        (* Switch: '<S1>/Switch2' incorporates:
         *  Constant: '<S1>/Constant3' *)

        IF Enable THEN 
            (* Switch: '<S1>/Switch3' incorporates:
             *  Constant: '<S1>/Constant3'
             *  Gain: '<S1>/Gain'
             *  Gain: '<S1>/Gain3'
             *  Gain: '<S1>/muC'
             *  Product: '<S1>/Product'
             *  Product: '<S1>/Product1'
             *  Sum: '<S1>/Add'
             *  Sum: '<S1>/Subtract'
             *  Sum: '<S1>/Subtract1' *)

            IF Clock > 0.01 THEN 
                uPF := ((((pAsimbar - pp) * 100000.0) - (((pBsimbar - pr) * 100000.0) * 0.7101)) * HPF_Num1) * kQf;
            ELSE 
                uPF := 0.0;
            END_IF;

            (* End of Switch: '<S1>/Switch3' *)
        ELSE 
            uPF := 0.0;
        END_IF;

        (* End of Switch: '<S1>/Switch2' *)
        

        (* Saturate: '<S1>/Saturation5' *)

        IF uPF >= 3600.0 THEN 
            uPF := 3600.0;
        ELSIF uPF <= -3600.0 THEN 
            uPF := -3600.0;
        END_IF;

        (* End of Saturate: '<S1>/Saturation5' *)
END_CASE;

END_FUNCTION_BLOCK

// IndraMotionMlc1/Application/SCC_Acceleration_Feedback
FUNCTION_BLOCK SCC_Acceleration_Feedback
VAR_INPUT
	ssMethodType: SINT;
	AF_on: BOOL;
	Direct_on: BOOL;
	LPF_on: BOOL;
	HPF_on: BOOL;
	Acc_Input: LREAL;
	D_rev: LREAL;
	K_Direct: LREAL;
	LPF_Num1: LREAL;
	LPF_Num2: LREAL;
	LPF_Den1: LREAL;
	LPF_Den2: LREAL;
	HPF_Num1: LREAL;
	HPF_Num2: LREAL;
	HPF_Den1: LREAL;
	HPF_Den2: LREAL;
	b_reset: BOOL;
END_VAR
VAR_OUTPUT
	u_Direct: LREAL;
	u_LPF: LREAL;
	u_HPF: LREAL;
	u_AF: LREAL;
END_VAR
VAR
	rtb_DiscreteTransferFcn: LREAL;
	rtb_DiscreteTransferFcn1: LREAL;
	rtb_bDirect: LREAL;
	rtb_bLPF: LREAL;
	rtb_bHPF: DINT;
	DiscreteTransferFcn_tmp: LREAL;
	tmp: BOOL;
	temp1: BOOL;
	temp2: BOOL;
	VectorConcatenate: ARRAY[0..1] OF LREAL;
	VectorConcatenate1: ARRAY[0..1] OF LREAL;
	VectorConcatenate2: ARRAY[0..1] OF LREAL;
	VectorConcatenate3: ARRAY[0..1] OF LREAL;
	DiscreteTransferFcn_states: LREAL;
	DiscreteTransferFcn1_states: LREAL;
END_VAR



CASE ssMethodType OF
    0: 
        (* SystemInitialize for Atomic SubSystem: '<Root>/SCC_Acceleration_Feedback' *)
        (* InitializeConditions for DiscreteTransferFcn: '<S1>/Discrete Transfer Fcn' *)
        DiscreteTransferFcn_states := 0.0;
        (* InitializeConditions for DiscreteTransferFcn: '<S1>/Discrete Transfer Fcn1' *)
        DiscreteTransferFcn1_states := 0.0;
        (* End of SystemInitialize for SubSystem: '<Root>/SCC_Acceleration_Feedback' *)
    1: 
        (* Outputs for Atomic SubSystem: '<Root>/SCC_Acceleration_Feedback' *)
        (* SignalConversion: '<S1>/ConcatBufferAtVector ConcatenateIn1' *)
        VectorConcatenate[0] := HPF_Num1;
        (* SignalConversion: '<S1>/ConcatBufferAtVector ConcatenateIn2' *)
        VectorConcatenate[1] := HPF_Num2;
        (* SignalConversion: '<S1>/ConcatBufferAtVector Concatenate1In1' *)
        VectorConcatenate1[0] := HPF_Den1;
        (* SignalConversion: '<S1>/ConcatBufferAtVector Concatenate1In2' *)
        VectorConcatenate1[1] := HPF_Den2;
        (* SignalConversion: '<S1>/ConcatBufferAtVector Concatenate2In1' *)
        VectorConcatenate2[0] := LPF_Num1;
        (* SignalConversion: '<S1>/ConcatBufferAtVector Concatenate2In2' *)
        VectorConcatenate2[1] := LPF_Num2;
        (* SignalConversion: '<S1>/ConcatBufferAtVector Concatenate3In1' *)
        VectorConcatenate3[0] := LPF_Den1;
        (* SignalConversion: '<S1>/ConcatBufferAtVector Concatenate3In2' *)
        VectorConcatenate3[1] := LPF_Den2;
        (* Product: '<S1>/Divide' incorporates:
         *  Gain: '<S1>/Unit Gain2'
         *  Product: '<S1>/Product' *)
        u_Direct := ((K_Direct * Acc_Input) * 6.0E+7) / D_rev;
        (* MATLAB Function: '<S1>/MATLAB Function' *)
        (* MATLAB Function 'SCC_Acceleration_Feedback/MATLAB Function': '<S2>:1' *)
        (* '<S2>:1:3' bDirect = 0; *)
        rtb_bDirect := 0.0;
        (* '<S2>:1:4' bLPF = 0; *)
        rtb_bLPF := 0.0;
        (* '<S2>:1:5' bHPF = 0; *)
        rtb_bHPF := 0;
        (* '<S2>:1:7' if Direct_on == 1 &amp;&amp; LPF_on == 0 &amp;&amp; HPF_on == 0 *)
        tmp :=  NOT HPF_on;
        temp2 :=  NOT LPF_on;

        IF (Direct_on AND temp2) AND tmp THEN 
            (* '<S2>:1:8' bDirect = 1; *)
            rtb_bDirect := 1.0;
        ELSE 
            temp1 :=  NOT Direct_on;

            IF (temp1 AND LPF_on) AND tmp THEN 
                (* '<S2>:1:9' elseif Direct_on == 0 &amp;&amp; LPF_on == 1 &amp;&amp; HPF_on == 0 *)
                (* '<S2>:1:10' bLPF = 1; *)
                rtb_bLPF := 1.0;
            ELSIF (temp1 AND temp2) AND HPF_on THEN 
                (* '<S2>:1:11' elseif Direct_on == 0 &amp;&amp; LPF_on == 0 &amp;&amp; HPF_on == 1 *)
                (* '<S2>:1:12' bHPF = 1; *)
                rtb_bHPF := 1;
            END_IF;

        END_IF;

        (* End of MATLAB Function: '<S1>/MATLAB Function' *)
        

        (* DiscreteTransferFcn: '<S1>/Discrete Transfer Fcn' incorporates:
         *  DiscreteTransferFcn: '<S1>/Discrete Transfer Fcn1' *)

        IF b_reset THEN 
            DiscreteTransferFcn_states := 0.0;
            DiscreteTransferFcn1_states := 0.0;
        END_IF;

        DiscreteTransferFcn_tmp := Acc_Input - (VectorConcatenate3[1] * DiscreteTransferFcn_states);
        (* Product: '<S1>/Divide1' incorporates:
         *  DiscreteTransferFcn: '<S1>/Discrete Transfer Fcn'
         *  Gain: '<S1>/Unit Gain' *)
        u_LPF := (((VectorConcatenate2[0] * DiscreteTransferFcn_tmp) + (VectorConcatenate2[1] * DiscreteTransferFcn_states)) * 6.0E+7) / D_rev;
        (* DiscreteTransferFcn: '<S1>/Discrete Transfer Fcn1' *)
        rtb_DiscreteTransferFcn := Acc_Input - (VectorConcatenate1[1] * DiscreteTransferFcn1_states);
        (* Product: '<S1>/Divide2' incorporates:
         *  DiscreteTransferFcn: '<S1>/Discrete Transfer Fcn1'
         *  Gain: '<S1>/Unit Gain1' *)
        u_HPF := (((VectorConcatenate[0] * rtb_DiscreteTransferFcn) + (VectorConcatenate[1] * DiscreteTransferFcn1_states)) * 6.0E+7) / D_rev;
        (* Switch: '<S1>/Switch' incorporates:
         *  Constant: '<S1>/Constant'
         *  Sum: '<S1>/Add' *)

        IF AF_on THEN 
            (* Switch: '<S1>/Switch3' incorporates:
             *  Constant: '<S1>/Constant' *)

            IF rtb_bHPF > 0 THEN 
                rtb_DiscreteTransferFcn1 := u_HPF;
            ELSE 
                rtb_DiscreteTransferFcn1 := 0.0;
            END_IF;

            (* End of Switch: '<S1>/Switch3' *)
            

            (* Switch: '<S1>/Switch2' *)

            IF rtb_bLPF > 0.0 THEN 
                rtb_bLPF := u_LPF;
            END_IF;

            (* End of Switch: '<S1>/Switch2' *)
            

            (* Switch: '<S1>/Switch1' *)

            IF rtb_bDirect > 0.0 THEN 
                rtb_bDirect := u_Direct;
            END_IF;

            (* End of Switch: '<S1>/Switch1' *)
            u_AF := (rtb_bDirect + rtb_bLPF) + rtb_DiscreteTransferFcn1;
        ELSE 
            u_AF := 0.0;
        END_IF;

        (* End of Switch: '<S1>/Switch' *)
        

        (* Saturate: '<S1>/Saturation' *)

        IF u_AF >= 3600.0 THEN 
            (* Outport: '<Root>/u_AF' *)
            u_AF := 3600.0;
        ELSIF u_AF <= -3600.0 THEN 
            (* Outport: '<Root>/u_AF' *)
            u_AF := -3600.0;
        END_IF;

        (* End of Saturate: '<S1>/Saturation' *)
        

        (* Update for DiscreteTransferFcn: '<S1>/Discrete Transfer Fcn' *)
        DiscreteTransferFcn_states := DiscreteTransferFcn_tmp;
        (* Update for DiscreteTransferFcn: '<S1>/Discrete Transfer Fcn1' *)
        DiscreteTransferFcn1_states := rtb_DiscreteTransferFcn;
        (* End of Outputs for SubSystem: '<Root>/SCC_Acceleration_Feedback' *)
END_CASE;

END_FUNCTION_BLOCK

// IndraMotionMlc1/Application/Delay_Vel
FUNCTION_BLOCK Delay_Vel
VAR_INPUT
	ssMethodType: SINT;
	Delay_ms: UDINT;
	Reset: BOOL;
	In: LREAL;
END_VAR
VAR_OUTPUT
	Out: LREAL;
END_VAR
VAR
	i: DINT;
	Delay_DSTATE: ARRAY[0..199] OF LREAL;
END_VAR



CASE ssMethodType OF
    0: 
        (* InitializeConditions for Delay: '<S1>/Delay' *)

        FOR i := 0 TO 199 DO 
            Delay_DSTATE[i] := 0.0;
        END_FOR;

        (* End of InitializeConditions for Delay: '<S1>/Delay' *)
    1: 
        (* Delay: '<S1>/Delay' *)

        IF Reset THEN 

            FOR i := 0 TO 199 DO 
                Delay_DSTATE[i] := 0.0;
            END_FOR;

        END_IF;


        IF Delay_ms <= 0 THEN 
            (* Outport: '<Root>/Out' *)
            Out := In;
        ELSE 

            IF Delay_ms > 200 THEN 
                i := 200;
            ELSE 
                i := UDINT_TO_DINT(Delay_ms);
            END_IF;

            (* Outport: '<Root>/Out' *)
            Out := Delay_DSTATE[200 - DINT_TO_UDINT(i)];
        END_IF;

        (* End of Delay: '<S1>/Delay' *)
        

        (* Update for Delay: '<S1>/Delay' *)

        FOR i := 0 TO 198 DO 
            Delay_DSTATE[i] := Delay_DSTATE[i + 1];
        END_FOR;

        Delay_DSTATE[199] := In;
        (* End of Update for Delay: '<S1>/Delay' *)
END_CASE;

END_FUNCTION_BLOCK

// IndraMotionMlc1/Application/Delay_Pos
FUNCTION_BLOCK Delay_Pos
VAR_INPUT
	ssMethodType: SINT;
	Delay_ms: UDINT;
	Initial_Pos_mm: LREAL;
	Reset: BOOL;
	In: LREAL;
END_VAR
VAR_OUTPUT
	Out: LREAL;
END_VAR
VAR
	i: DINT;
	icLoad: USINT;
	Delay_DSTATE: ARRAY[0..199] OF LREAL;
END_VAR



CASE ssMethodType OF
    0: 
        (* InitializeConditions for Delay: '<S1>/Delay' *)
        icLoad := 1;
    1: 
        (* Delay: '<S1>/Delay' *)

        IF Reset THEN 
            icLoad := 1;
        END_IF;


        IF icLoad <> 0 THEN 

            FOR i := 0 TO 199 DO 
                Delay_DSTATE[i] := Initial_Pos_mm;
            END_FOR;

        END_IF;


        IF Delay_ms <= 0 THEN 
            (* Outport: '<Root>/Out' *)
            Out := In;
        ELSE 

            IF Delay_ms > 200 THEN 
                i := 200;
            ELSE 
                i := UDINT_TO_DINT(Delay_ms);
            END_IF;

            (* Outport: '<Root>/Out' *)
            Out := Delay_DSTATE[200 - DINT_TO_UDINT(i)];
        END_IF;

        (* End of Delay: '<S1>/Delay' *)
        

        (* Update for Delay: '<S1>/Delay' *)
        icLoad := 0;

        FOR i := 0 TO 198 DO 
            Delay_DSTATE[i] := Delay_DSTATE[i + 1];
        END_FOR;

        Delay_DSTATE[199] := In;
        (* End of Update for Delay: '<S1>/Delay' *)
END_CASE;

END_FUNCTION_BLOCK

// IndraMotionMlc1/Application/SCC_VFF
FUNCTION_BLOCK SCC_VFF
VAR_INPUT
	VFF_On: BOOL;
	kVFF: LREAL;
	Aa: LREAL;
	kq: LREAL;
	v_ref_mms: LREAL;
END_VAR
VAR_OUTPUT
	uFF: LREAL;
END_VAR
VAR
END_VAR


(* Switch: '<S1>/Switch1' *)

IF VFF_On THEN 
    (* Outport: '<Root>/uFF' incorporates:
     *  Gain: '<S1>/Gain1'
     *  Product: '<S1>/Divide1'
     *  Product: '<S1>/Product'
     *  Product: '<S1>/Product1' *)
    uFF := (((0.001 * v_ref_mms) * Aa) / kq) * kVFF;
ELSE 
    (* Outport: '<Root>/uFF' incorporates:
     *  Constant: '<S1>/Constant' *)
    uFF := 0.0;
END_IF;

(* End of Switch: '<S1>/Switch1' *)

END_FUNCTION_BLOCK

// IndraMotionMlc1/Application/SCC_Controller_PFB1
FUNCTION_BLOCK SCC_Controller_PFB1
VAR_INPUT
	ssMethodType: SINT;
	PFB_On: BOOL;
	Int_On: BOOL;
	k_P: LREAL;
	k_I: LREAL;
	Pos_Ref_mm: LREAL;
	Pos_FB_mm: LREAL;
	Reset_I_ctrl: BOOL;
END_VAR
VAR_OUTPUT
	uPFB: LREAL;
	u_I_ctrl: LREAL;
	Pos_Error: LREAL;
END_VAR
VAR
	rtb_Switch2: LREAL;
	rtb_u_FB: LREAL;
	c_DiscreteTimeIntegrator_DS: LREAL;
END_VAR



CASE ssMethodType OF
    0: 
        (* InitializeConditions for DiscreteIntegrator: '<S1>/Discrete-Time Integrator' *)
        c_DiscreteTimeIntegrator_DS := 0.0;
    1: 
        (* Switch: '<S1>/Switch2' *)

        IF Reset_I_ctrl THEN 
            (* DiscreteIntegrator: '<S1>/Discrete-Time Integrator' *)
            c_DiscreteTimeIntegrator_DS := 0.0;
        END_IF;

        (* End of Switch: '<S1>/Switch2' *)
        

        (* Sum: '<S1>/Sum1' incorporates:
         *  Gain: '<S1>/Gain1'
         *  Gain: '<S1>/Gain2' *)
        rtb_Switch2 := (0.001 * Pos_Ref_mm) - (0.001 * Pos_FB_mm);
        (* Switch: '<S1>/Switch' incorporates:
         *  Constant: '<S1>/Constant'
         *  DiscreteIntegrator: '<S1>/Discrete-Time Integrator' *)

        IF Int_On THEN 
            u_I_ctrl := c_DiscreteTimeIntegrator_DS;
        ELSE 
            u_I_ctrl := 0.0;
        END_IF;

        (* End of Switch: '<S1>/Switch' *)
        

        (* Sum: '<S1>/Sum5' incorporates:
         *  Product: '<S1>/Product' *)
        rtb_u_FB := (k_P * rtb_Switch2) + u_I_ctrl;
        (* Saturate: '<S1>/Saturation1' *)

        IF rtb_u_FB >= 3200.0 THEN 
            uPFB := 3200.0;
        ELSIF rtb_u_FB > -3200.0 THEN 
            uPFB := rtb_u_FB;
        ELSE 
            uPFB := -3200.0;
        END_IF;

        (* End of Saturate: '<S1>/Saturation1' *)
        

        (* Sum: '<S1>/Sum3' *)
        rtb_u_FB := uPFB - rtb_u_FB;
        (* Switch: '<S1>/Switch1' incorporates:
         *  Constant: '<S1>/Constant1' *)

        IF  NOT PFB_On THEN 
            uPFB := 0.0;
        END_IF;

        (* End of Switch: '<S1>/Switch1' *)
        

        (* Outport: '<Root>/Pos_Error' incorporates:
         *  Gain: '<S1>/Gain3' *)
        Pos_Error := -1000.0 * rtb_Switch2;
        (* Update for DiscreteIntegrator: '<S1>/Discrete-Time Integrator' incorporates:
         *  Product: '<S1>/Divide'
         *  Product: '<S1>/Product2'
         *  Sum: '<S1>/Sum2' *)
        c_DiscreteTimeIntegrator_DS := ((((rtb_u_FB / k_P) + rtb_Switch2) * k_I) * 0.001) + c_DiscreteTimeIntegrator_DS;
END_CASE;

END_FUNCTION_BLOCK

// IndraMotionMlc1/Application/SCC_Ramp_Test
FUNCTION_BLOCK SCC_Ramp_Test
VAR_INPUT
	Enable: BOOL;
	n0: LREAL;
	nExt: LREAL;
	nRetr: LREAL;
	t0: LREAL;
	tRampUp: LREAL;
	tHold: LREAL;
	tRampDown: LREAL;
	tWait: LREAL;
	CyclicTime: LREAL;
END_VAR
VAR_OUTPUT
	uEM: LREAL;
	T: LREAL;
END_VAR
VAR
	slopeExt: LREAL;
	slopeRetr: LREAL;
	tmp: LREAL;
	temp1: LREAL;
END_VAR


(* MATLAB Function: '<S1>/WaveSignal' *)
(* MATLAB Function 'SCC_Ramp_Test/WaveSignal': '<S2>:1' *)
(* '<S2>:1:2' slopeExt=u0-uExt; *)
slopeExt := n0 - nExt;
(* '<S2>:1:3' slopeRetr=uRetr-u0; *)
slopeRetr := nRetr - n0;
(* '<S2>:1:4' t1=tRampUp; *)
(* '<S2>:1:5' t2=tHold; *)
(* '<S2>:1:6' t3=tRampDown; *)
(* '<S2>:1:7' t4=tWait; *)
(* '<S2>:1:8' t5=t1; *)
(* '<S2>:1:9' t6=t2; *)
(* '<S2>:1:10' t7=t3; *)
(* '<S2>:1:12' if t>=0 &amp;&amp; t<t0 *)

IF (CyclicTime >= 0.0) AND (CyclicTime < t0) THEN 
    (* '<S2>:1:13' u = u0; *)
    uEM := n0;
ELSE 
    tmp := t0 + tRampUp;

    IF (CyclicTime >= t0) AND (CyclicTime < tmp) THEN 
        (* '<S2>:1:14' elseif t>=t0 &amp;&amp; t<(t0+t1) *)
        (* '<S2>:1:15' u = u0-(slopeExt/t1)*(t-t0); *)
        uEM := n0 - ((slopeExt / tRampUp) * (CyclicTime - t0));
    ELSE 
        temp1 := tmp + tHold;

        IF (CyclicTime >= tmp) AND (CyclicTime < temp1) THEN 
            (* '<S2>:1:16' elseif t>=(t0+t1) &amp;&amp; t<(t0+t1+t2) *)
            (* '<S2>:1:17' u = uExt; *)
            uEM := nExt;
        ELSE 
            tmp := temp1 + tRampDown;

            IF (CyclicTime >= temp1) AND (CyclicTime < tmp) THEN 
                (* '<S2>:1:18' elseif t>=(t0+t1+t2) &amp;&amp; t<(t0+t1+t2+t3) *)
                (* '<S2>:1:19' u = uExt+(slopeExt/t3)*(t-(t0+t1+t2)); *)
                uEM := ((CyclicTime - temp1) * (slopeExt / tRampDown)) + nExt;
            ELSE 
                temp1 := tmp + tWait;

                IF (CyclicTime >= tmp) AND (CyclicTime < temp1) THEN 
                    (* '<S2>:1:20' elseif t>=(t0+t1+t2+t3) &amp;&amp; t<(t0+t1+t2+t3+t4) *)
                    (* '<S2>:1:21' u = u0; *)
                    uEM := n0;
                ELSE 
                    tmp := temp1 + tRampUp;

                    IF (CyclicTime >= temp1) AND (CyclicTime < tmp) THEN 
                        (* '<S2>:1:22' elseif t>=(t0+t1+t2+t3+t4) &amp;&amp; t<(t0+t1+t2+t3+t4+t5) *)
                        (* '<S2>:1:23' u = u0+(slopeRetr/t5)*(t-(t0+t1+t2+t3+t4)); *)
                        uEM := ((CyclicTime - temp1) * (slopeRetr / tRampUp)) + n0;
                    ELSE 
                        temp1 := tmp + tHold;

                        IF (CyclicTime >= tmp) AND (CyclicTime < temp1) THEN 
                            (* '<S2>:1:24' elseif t>=(t0+t1+t2+t3+t4+t5) &amp;&amp; t<(t0+t1+t2+t3+t4+t5+t6) *)
                            (* '<S2>:1:25' u = uRetr; *)
                            uEM := nRetr;
                        ELSIF (CyclicTime >= temp1) AND (CyclicTime < (temp1 + tRampDown)) THEN 
                            (* '<S2>:1:26' elseif t>=(t0+t1+t2+t3+t4+t5+t6) &amp;&amp; t<(t0+t1+t2+t3+t4+t5+t6+t7) *)
                            (* '<S2>:1:27' u = uRetr-(slopeRetr/t3)*(t-(t0+t1+t2+t3+t4+t5+t6)); *)
                            uEM := nRetr - ((CyclicTime - temp1) * (slopeRetr / tRampDown));
                        ELSE 
                            (* '<S2>:1:28' else *)
                            (* '<S2>:1:29' u = u0; *)
                            uEM := n0;
                        END_IF;

                    END_IF;

                END_IF;

            END_IF;

        END_IF;

    END_IF;

END_IF;

(* Switch: '<S1>/Switch' *)
(* '<S2>:1:32' T = t0+t1+t2+t3+t4+t5+t6+t7; *)

IF  NOT Enable THEN 
    (* Outport: '<Root>/uEM' *)
    uEM := n0;
END_IF;

(* End of Switch: '<S1>/Switch' *)


(* Outport: '<Root>/T' incorporates:
 *  MATLAB Function: '<S1>/WaveSignal' *)
T := ((((((t0 + tRampUp) + tHold) + tRampDown) + tWait) + tRampUp) + tHold) + tRampDown;

END_FUNCTION_BLOCK

// IndraMotionMlc1/Application/LHV_Controller2
FUNCTION_BLOCK LHV_Controller2
VAR_INPUT
	LHC_On: BOOL;
	Enabler: BOOL;
	kP: LREAL;
	p_3: LREAL;
	p_1: LREAL;
END_VAR
VAR_OUTPUT
	error_bar: LREAL;
	Out_rpm: LREAL;
END_VAR
VAR
	rtb_u: LREAL;
END_VAR


(* Switch: '<S1>/Switch6' incorporates:
 *  Constant: '<S1>/Constant7' *)

IF Enabler THEN 
    Out_rpm := p_1;
ELSE 
    Out_rpm := 0.0;
END_IF;

(* End of Switch: '<S1>/Switch6' *)


(* Gain: '<S1>/1' *)
rtb_u := 100000.0 * Out_rpm;
(* Switch: '<S1>/Switch5' incorporates:
 *  Constant: '<S1>/Constant7' *)

IF Enabler THEN 
    Out_rpm := p_3;
ELSE 
    Out_rpm := 0.0;
END_IF;

(* End of Switch: '<S1>/Switch5' *)


(* Switch: '<S1>/Switch1' incorporates:
 *  Constant: '<S1>/Constant'
 *  Gain: '<S1>/12'
 *  Gain: '<S1>/Gain15'
 *  Product: '<S1>/Product'
 *  Sum: '<S1>/Add6' *)

IF LHC_On THEN 
    Out_rpm := (((100000.0 * Out_rpm) - rtb_u) * kP) * 9.5492965855137211;
ELSE 
    Out_rpm := 0.0;
END_IF;

(* End of Switch: '<S1>/Switch1' *)


(* Saturate: '<S1>/Saturation1' *)

IF Out_rpm >= 1000.0 THEN 
    Out_rpm := 1000.0;
ELSIF Out_rpm <= -1000.0 THEN 
    Out_rpm := -1000.0;
END_IF;

(* End of Saturate: '<S1>/Saturation1' *)


(* Outport: '<Root>/error_bar ' incorporates:
 *  Sum: '<S1>/Add1' *)
error_bar := p_3 - p_1;

END_FUNCTION_BLOCK

// IndraMotionMlc1/Application/CC_PI_FF_AD
FUNCTION_BLOCK CC_PI_FF_AD
VAR_INPUT
	ssMethodType: SINT;
	Enable: BOOL;
	FB_controller_ON: LREAL;
	I_controller_ON: LREAL;
	ActiveLH_ON: LREAL;
	kP: LREAL;
	kI: LREAL;
	MaxError: LREAL;
	Pos_Ref: LREAL;
	Vel_Ref: LREAL;
	PosFeedBack: LREAL;
	p001: LREAL;
	p009: LREAL;
END_VAR
VAR_OUTPUT
	nRef: LREAL;
	PosError: LREAL;
	LHenable: BOOL;
END_VAR
VAR
	rtb_x1: LREAL;
	rtb_Switch1: DINT;
	rtb_FBcontrollerLimiter: LREAL;
	rtb_Enabler: DINT;
	rtb_LoadPressure: LREAL;
	TransferFcn1_tmp: LREAL;
	c_DiscreteTimeIntegrator_DS: LREAL;
	TransferFcn1_states: LREAL;
END_VAR



CASE ssMethodType OF
    0: 
        (* InitializeConditions for DiscreteIntegrator: '<S1>/Discrete-Time Integrator' *)
        c_DiscreteTimeIntegrator_DS := 0.0;
        (* InitializeConditions for DiscreteTransferFcn: '<S1>/Transfer Fcn1 ' *)
        TransferFcn1_states := 0.0;
    1: 
        (* Sum: '<S1>/Sum' *)
        PosError := Pos_Ref - PosFeedBack;
        (* MATLAB Function: '<S1>/MATLAB Function3' incorporates:
         *  MATLAB Function: '<S1>/MATLAB Function'
         *  MATLAB Function: '<S1>/MATLAB Function2' *)
        (* MATLAB Function 'CC_PI_FF_AD/MATLAB Function3': '<S5>:1' *)
        (* '<S5>:1:3' if  abs(cmd) > 0.005 *)
        TransferFcn1_tmp := ABS(Vel_Ref);

        IF TransferFcn1_tmp > 0.005 THEN 
            (* '<S5>:1:4' Enabler = 1; *)
            rtb_Enabler := 1;
        ELSIF ABS(PosError) > MaxError THEN 
            (* '<S5>:1:5' elseif abs(error) > MaxError *)
            (* '<S5>:1:6' Enabler = 1; *)
            rtb_Enabler := 1;
        ELSE 
            (* '<S5>:1:7' else *)
            (* '<S5>:1:8' Enabler = 0; *)
            rtb_Enabler := 0;
        END_IF;

        (* End of MATLAB Function: '<S1>/MATLAB Function3' *)
        

        (* Switch: '<S1>/Switch5' incorporates:
         *  Constant: '<S1>/Constant5' *)

        IF  NOT (ActiveLH_ON > 0.0) THEN 
            rtb_Enabler := 1;
        END_IF;

        (* End of Switch: '<S1>/Switch5' *)
        

        (* MATLAB Function: '<S1>/MATLAB Function' *)
        (* MATLAB Function 'CC_PI_FF_AD/MATLAB Function': '<S3>:1' *)
        (* '<S3>:1:3' if  abs(cmd) > 0.005 *)

        IF TransferFcn1_tmp > 0.005 THEN 
            (* '<S3>:1:4' x1 = 0; *)
            rtb_x1 := 0.0;
        ELSIF ABS(PosError) > MaxError THEN 
            (* '<S3>:1:5' elseif abs(error) > MaxError *)
            (* '<S3>:1:6' x1 = 0; *)
            rtb_x1 := 0.0;
        ELSE 
            (* '<S3>:1:7' else *)
            (* '<S3>:1:8' x1 = 1; *)
            rtb_x1 := 1.0;
        END_IF;

        (* Switch: '<S1>/Switch1' incorporates:
         *  Constant: '<S1>/Constant1'
         *  Constant: '<S1>/Constant2'
         *  DataTypeConversion: '<S1>/Data Type Conversion1' *)

        IF rtb_x1 <> 0.0 THEN 
            rtb_Switch1 := 1;
        ELSE 
            rtb_Switch1 := 0;
        END_IF;

        (* End of Switch: '<S1>/Switch1' *)
        

        (* DiscreteIntegrator: '<S1>/Discrete-Time Integrator' *)

        IF rtb_Switch1 <> 0 THEN 
            c_DiscreteTimeIntegrator_DS := 0.0;
        END_IF;

        (* Switch: '<S1>/Switch4' incorporates:
         *  Constant: '<S1>/Constant4'
         *  DiscreteIntegrator: '<S1>/Discrete-Time Integrator' *)

        IF I_controller_ON > 0.0 THEN 
            rtb_x1 := c_DiscreteTimeIntegrator_DS;
        ELSE 
            rtb_x1 := 0.0;
        END_IF;

        (* End of Switch: '<S1>/Switch4' *)
        

        (* Sum: '<S1>/Sum1' incorporates:
         *  Product: '<S1>/Product1' *)
        rtb_x1 := (PosError * kP) + rtb_x1;
        (* Saturate: '<S1>/FB controller Limiter' *)

        IF rtb_x1 >= 3500.0 THEN 
            rtb_FBcontrollerLimiter := 3500.0;
        ELSIF rtb_x1 > -3500.0 THEN 
            rtb_FBcontrollerLimiter := rtb_x1;
        ELSE 
            rtb_FBcontrollerLimiter := -3500.0;
        END_IF;

        (* End of Saturate: '<S1>/FB controller Limiter' *)
        

        (* MATLAB Function: '<S1>/MATLAB Function2' incorporates:
         *  DataTypeConversion: '<S1>/Data Type Conversion' *)
        (* MATLAB Function 'CC_PI_FF_AD/MATLAB Function2': '<S4>:1' *)
        (* '<S4>:1:3' if  abs(cmd) > 0.005 &amp;&amp; LHenable > 0 *)

        IF (TransferFcn1_tmp > 0.005) AND (rtb_Enabler <> 0) THEN 
            (* '<S4>:1:4' Enabler = 1; *)
            rtb_Switch1 := 1;
        ELSIF ABS(PosError) > MaxError THEN 

            IF rtb_Enabler <> 0 THEN 
                (* '<S4>:1:5' elseif abs(error) > MaxError &amp;&amp; LHenable > 0 *)
                (* '<S4>:1:6' Enabler = 1; *)
                rtb_Switch1 := 1;
            ELSE 
                (* '<S4>:1:7' else *)
                (* '<S4>:1:8' Enabler = 0; *)
                rtb_Switch1 := 0;
            END_IF;

        ELSE 
            (* '<S4>:1:7' else *)
            (* '<S4>:1:8' Enabler = 0; *)
            rtb_Switch1 := 0;
        END_IF;

        (* DiscreteTransferFcn: '<S1>/Transfer Fcn1 ' incorporates:
         *  Gain: '<S1>/Cylinder Area Ratio'
         *  Gain: '<S1>/Gain'
         *  Gain: '<S1>/Gain1'
         *  Sum: '<S1>/Load Pressure' *)
        TransferFcn1_tmp := ((100000.0 * p001) - ((100000.0 * p009) * 0.710059171597633)) - (-0.997 * TransferFcn1_states);
        (* Switch: '<S1>/Switch6' *)

        IF Enable THEN 
            (* Switch: '<S1>/Switch3' incorporates:
             *  Constant: '<S1>/Constant3' *)

            IF rtb_Switch1 > 0 THEN 
                (* Switch: '<S1>/Switch2' incorporates:
                 *  Constant: '<S1>/Constant' *)

                IF FB_controller_ON > 0.0 THEN 
                    rtb_LoadPressure := rtb_FBcontrollerLimiter;
                ELSE 
                    rtb_LoadPressure := 0.0;
                END_IF;

                (* End of Switch: '<S1>/Switch2' *)
                

                (* Switch: '<S2>/Switch' incorporates:
                 *  Gain: '<S2>/Lift crane (pumping mode)'
                 *  Gain: '<S2>/Lower crane (motoring mode)' *)

                IF Vel_Ref >= 0.0 THEN 
                    nRef := 19.7715 * Vel_Ref;
                ELSE 
                    nRef := 17.8438 * Vel_Ref;
                END_IF;

                (* End of Switch: '<S2>/Switch' *)
                

                (* Sum: '<S1>/Sum9' incorporates:
                 *  DiscreteTransferFcn: '<S1>/Transfer Fcn1 ' *)
                nRef := (nRef + rtb_LoadPressure) - ((5.0E-5 * TransferFcn1_tmp) + (-5.0E-5 * TransferFcn1_states));
                (* Saturate: '<S1>/Rev limiter for motor +//- 3000 [rpm]' *)

                IF nRef >= 3500.0 THEN 
                    nRef := 3500.0;
                ELSIF  NOT (nRef > -3500.0) THEN 
                    nRef := -3500.0;
                END_IF;

                (* End of Saturate: '<S1>/Rev limiter for motor +//- 3000 [rpm]' *)
            ELSE 
                nRef := 0.0;
            END_IF;

            (* End of Switch: '<S1>/Switch3' *)
        ELSE 
            (* Outport: '<Root>/nRef' incorporates:
             *  Constant: '<S1>/Constant6' *)
            nRef := 0.0;
        END_IF;

        (* End of Switch: '<S1>/Switch6' *)
        

        (* Outport: '<Root>/LHenable' incorporates:
         *  DataTypeConversion: '<S1>/Data Type Conversion' *)
        LHenable := rtb_Enabler <> 0;
        (* Update for DiscreteIntegrator: '<S1>/Discrete-Time Integrator' incorporates:
         *  Product: '<S1>/Divide'
         *  Product: '<S1>/Product'
         *  Sum: '<S1>/Sum2'
         *  Sum: '<S1>/Sum3' *)
        c_DiscreteTimeIntegrator_DS := (((((rtb_FBcontrollerLimiter - rtb_x1) / kP) + PosError) * kI) * 0.001) + c_DiscreteTimeIntegrator_DS;
        (* Update for DiscreteTransferFcn: '<S1>/Transfer Fcn1 ' *)
        TransferFcn1_states := TransferFcn1_tmp;
END_CASE;

END_FUNCTION_BLOCK

// IndraMotionMlc1/Application/SCC_Controller_FF_PI_AD
FUNCTION_BLOCK SCC_Controller_FF_PI_AD
VAR_INPUT
	ssMethodType: SINT;
	Enable: BOOL;
	LH_Active_On: BOOL;
	Tuning_Mode_On: BOOL;
	FB_Cntr_On: BOOL;
	I_Cntr_On: BOOL;
	I_Cntr_Reset_On: BOOL;
	Active_Damper_On: BOOL;
	k_AD_Num: LREAL;
	Pos_Error_Limit: LREAL;
	k_FF_Up: LREAL;
	k_FF_Down: LREAL;
	k_P: LREAL;
	k_I: LREAL;
	Pos_Ref: LREAL;
	Vel_Ref: LREAL;
	Pos_FB: LREAL;
	p_A: LREAL;
	p_B: LREAL;
END_VAR
VAR_OUTPUT
	Pos_Error: LREAL;
	u_FF: LREAL;
	u_P: LREAL;
	u_I: LREAL;
	u_AD: LREAL;
	I_reset: LREAL;
	n_Ref: LREAL;
	LH_Enable: BOOL;
END_VAR
VAR
	rtb_u_FB: LREAL;
	rtb_LoadPressure: LREAL;
	TransferFcn11_tmp: LREAL;
	VectorConcatenate: ARRAY[0..1] OF LREAL;
	c_DiscreteTimeIntegrator_DS: LREAL;
	TransferFcn11_states: LREAL;
END_VAR



CASE ssMethodType OF
    0: 
        (* InitializeConditions for DiscreteTransferFcn: '<S5>/Transfer Fcn1 1' *)
        TransferFcn11_states := 0.0;
        (* InitializeConditions for DiscreteIntegrator: '<S1>/Discrete-Time Integrator' *)
        c_DiscreteTimeIntegrator_DS := 0.0;
    1: 
        (* Switch: '<S2>/Switch' incorporates:
         *  Product: '<S2>/Lift crane (pumping mode)'
         *  Product: '<S2>/Lower crane (motoring mode)' *)

        IF Vel_Ref >= 0.0 THEN 
            u_FF := k_FF_Up * Vel_Ref;
        ELSE 
            u_FF := Vel_Ref * k_FF_Down;
        END_IF;

        (* End of Switch: '<S2>/Switch' *)
        

        (* SignalConversion: '<S5>/ConcatBufferAtVector ConcatenateIn1' *)
        VectorConcatenate[0] := k_AD_Num;
        (* Gain: '<S5>/Gain1' *)
        VectorConcatenate[1] :=  -k_AD_Num;
        (* DiscreteTransferFcn: '<S5>/Transfer Fcn1 1' incorporates:
         *  Gain: '<S5>/Cylinder Area Ratio'
         *  Sum: '<S5>/Load Pressure' *)
        TransferFcn11_tmp := (p_A - (0.710059171597633 * p_B)) - (-0.997 * TransferFcn11_states);
        u_AD := (VectorConcatenate[0] * TransferFcn11_tmp) + (VectorConcatenate[1] * TransferFcn11_states);
        (* Sum: '<S1>/Sum1' *)
        Pos_Error := Pos_Ref - Pos_FB;
        (* MATLAB Function: '<S1>/From Jespers SimX1' *)
        (* MATLAB Function 'SCC_Controller_FF_PI_AD/From Jespers SimX1': '<S3>:1' *)
        (* '<S3>:1:3' I_Reset = 1; *)
        (* '<S3>:1:5' if (abs(Pos_Error) <= Pos_Error_Limit) &amp;&amp; (Vel_SP == 0) *)

        IF ABS(Pos_Error) <= Pos_Error_Limit THEN 

            IF Vel_Ref = 0.0 THEN 
                (* '<S3>:1:6' I_Reset = 1; *)
                rtb_LoadPressure := 1.0;
            ELSE 
                (* '<S3>:1:7' else *)
                (* '<S3>:1:8' I_Reset = 0; *)
                rtb_LoadPressure := 0.0;
            END_IF;

        ELSE 
            (* '<S3>:1:7' else *)
            (* '<S3>:1:8' I_Reset = 0; *)
            rtb_LoadPressure := 0.0;
        END_IF;

        (* End of MATLAB Function: '<S1>/From Jespers SimX1' *)
        

        (* Switch: '<S1>/Switch3' incorporates:
         *  Constant: '<S1>/Constant2' *)

        IF I_Cntr_Reset_On THEN 
            I_reset := rtb_LoadPressure;
        ELSE 
            I_reset := 0.0;
        END_IF;

        (* End of Switch: '<S1>/Switch3' *)
        

        (* DiscreteIntegrator: '<S1>/Discrete-Time Integrator' *)

        IF I_reset <> 0.0 THEN 
            c_DiscreteTimeIntegrator_DS := 0.0;
        END_IF;

        (* Product: '<S1>/Product' *)
        u_P := k_P * Pos_Error;
        (* Switch: '<S1>/Switch' incorporates:
         *  Constant: '<S1>/Constant'
         *  DiscreteIntegrator: '<S1>/Discrete-Time Integrator' *)

        IF I_Cntr_On THEN 
            u_I := c_DiscreteTimeIntegrator_DS;
        ELSE 
            u_I := 0.0;
        END_IF;

        (* End of Switch: '<S1>/Switch' *)
        

        (* Sum: '<S1>/Sum5' *)
        rtb_u_FB := u_P + u_I;
        (* Saturate: '<S1>/Saturation1' *)

        IF rtb_u_FB >= 3500.0 THEN 
            n_Ref := 3500.0;
        ELSIF rtb_u_FB > -3500.0 THEN 
            n_Ref := rtb_u_FB;
        ELSE 
            n_Ref := -3500.0;
        END_IF;

        (* End of Saturate: '<S1>/Saturation1' *)
        

        (* Sum: '<S1>/Sum3' *)
        rtb_u_FB := n_Ref - rtb_u_FB;
        (* Switch: '<S1>/Switch1' incorporates:
         *  Constant: '<S1>/Constant1' *)

        IF  NOT FB_Cntr_On THEN 
            n_Ref := 0.0;
        END_IF;

        (* End of Switch: '<S1>/Switch1' *)
        

        (* Switch: '<S1>/Switch4' incorporates:
         *  Constant: '<S1>/Constant3' *)

        IF  NOT Active_Damper_On THEN 
            u_AD := 0.0;
        END_IF;

        (* End of Switch: '<S1>/Switch4' *)
        

        (* Sum: '<S1>/Sum6' *)
        n_Ref := (u_FF + n_Ref) - u_AD;
        (* Saturate: '<S1>/Saturation2' *)

        IF n_Ref >= 3500.0 THEN 
            n_Ref := 3500.0;
        ELSIF  NOT (n_Ref > -3500.0) THEN 
            n_Ref := -3500.0;
        END_IF;

        (* End of Saturate: '<S1>/Saturation2' *)
        

        (* MATLAB Function: '<S1>/Motor Speed Ref' *)
        (* MATLAB Function 'SCC_Controller_FF_PI_AD/Motor Speed Ref': '<S4>:1' *)
        (* '<S4>:1:4' n_Motor = 0; *)
        (* '<S4>:1:6' if Enable == 0 *)

        IF  NOT Enable THEN 
            (* Outport: '<Root>/n_Ref' *)
            (* '<S4>:1:7' n_Motor = 0; *)
            n_Ref := 0.0;
        ELSIF ( NOT (rtb_LoadPressure = 0.0)) AND ( NOT Tuning_Mode_On) THEN 
            (* Outport: '<Root>/n_Ref' *)
            (* '<S4>:1:12' else *)
            (* '<S4>:1:13' n_Motor = 0; *)
            n_Ref := 0.0;
        END_IF;

        (* End of MATLAB Function: '<S1>/Motor Speed Ref' *)
        

        (* Switch: '<S1>/Switch5' *)

        IF LH_Active_On THEN 
            (* Switch: '<S1>/Switch2' *)

            IF rtb_LoadPressure > 0.0 THEN 
                (* Outport: '<Root>/LH_Enable' incorporates:
                 *  Constant: '<S1>/Constant4' *)
                LH_Enable := FALSE;
            ELSE 
                (* Outport: '<Root>/LH_Enable' incorporates:
                 *  Constant: '<S1>/Constant6' *)
                LH_Enable := TRUE;
            END_IF;

            (* End of Switch: '<S1>/Switch2' *)
        ELSE 
            (* Outport: '<Root>/LH_Enable' incorporates:
             *  Constant: '<S1>/Constant5' *)
            LH_Enable := TRUE;
        END_IF;

        (* End of Switch: '<S1>/Switch5' *)
        

        (* Update for DiscreteTransferFcn: '<S5>/Transfer Fcn1 1' *)
        TransferFcn11_states := TransferFcn11_tmp;
        (* Update for DiscreteIntegrator: '<S1>/Discrete-Time Integrator' incorporates:
         *  Product: '<S1>/Divide'
         *  Product: '<S1>/Product2'
         *  Sum: '<S1>/Sum2' *)
        c_DiscreteTimeIntegrator_DS := ((((rtb_u_FB / k_P) + Pos_Error) * k_I) * 0.001) + c_DiscreteTimeIntegrator_DS;
END_CASE;

END_FUNCTION_BLOCK

// IndraMotionMlc1/Application/Step_Damiano
FUNCTION_BLOCK Step_Damiano
VAR_INPUT
	n_SP: LREAL;
	CyclicTime: LREAL;
	t0: LREAL;
	t1: LREAL;
	t2: LREAL;
	t3: LREAL;
	t4: LREAL;
	LH_Activate: BOOL;
END_VAR
VAR_OUTPUT
	EndTime: LREAL;
	n_ref: LREAL;
	u_LH: BOOL;
END_VAR
VAR
	tmp: LREAL;
	temp1: LREAL;
END_VAR


(* MATLAB Function: '<S1>/StepFunction' *)
(* MATLAB Function 'Step_Damiano/StepFunction': '<S2>:1' *)
(* '<S2>:1:3' y = 0; *)
(* '<S2>:1:5' if t>=0 &amp;&amp; t<t0 *)

IF (CyclicTime >= 0.0) AND (CyclicTime < t0) THEN 
    (* Outport: '<Root>/n_ref' *)
    (* '<S2>:1:6' y = 0; *)
    n_ref := 0.0;
ELSE 
    tmp := t0 + t1;

    IF (CyclicTime >= t0) AND (CyclicTime < tmp) THEN 
        (* Outport: '<Root>/n_ref' *)
        (* '<S2>:1:7' elseif t>=(t0) &amp;&amp; t<(t0+t1) *)
        (* '<S2>:1:8' y = n_SP; *)
        n_ref := n_SP;
    ELSE 
        temp1 := tmp + t2;

        IF (CyclicTime >= tmp) AND (CyclicTime < temp1) THEN 
            (* Outport: '<Root>/n_ref' *)
            (* '<S2>:1:9' elseif t>=(t0+t1) &amp;&amp; t<(t0+t1+t2) *)
            (* '<S2>:1:10' y = 0; *)
            n_ref := 0.0;
        ELSE 
            tmp := temp1 + t3;

            IF (CyclicTime >= temp1) AND (CyclicTime < tmp) THEN 
                (* Outport: '<Root>/n_ref' *)
                (* '<S2>:1:11' elseif t>=(t0+t1+t2) &amp;&amp; t<(t0+t1+t2+t3) *)
                (* '<S2>:1:12' y = -n_SP; *)
                n_ref :=  -n_SP;
            ELSIF (CyclicTime >= tmp) AND (CyclicTime < (tmp + t4)) THEN 
                (* Outport: '<Root>/n_ref' *)
                (* '<S2>:1:13' elseif t>=(t0+t1+t2+t3) &amp;&amp; t<(t0+t1+t2+t3+t4) *)
                (* '<S2>:1:14' y = 0; *)
                n_ref := 0.0;
            ELSE 
                (* Outport: '<Root>/n_ref' *)
                (* '<S2>:1:15' else *)
                (* '<S2>:1:16' y = 0; *)
                n_ref := 0.0;
            END_IF;

        END_IF;

    END_IF;

END_IF;

(* Outport: '<Root>/EndTime' incorporates:
 *  MATLAB Function: '<S1>/StepFunction' *)
(* '<S2>:1:19' T = t0+t1+t2+t3+t4; *)
EndTime := (((t0 + t1) + t2) + t3) + t4;
(* Outport: '<Root>/u_LH' *)
u_LH := LH_Activate;

END_FUNCTION_BLOCK

// IndraMotionMlc1/Application/SCC_HPPF
FUNCTION_BLOCK SCC_HPPF
VAR_INPUT
	ssMethodType: SINT;
	Enable: BOOL;
	usDelay: LREAL;
	kQf: LREAL;
	HPF_Num1: LREAL;
	HPF_Num2: LREAL;
	HPF_Den1: LREAL;
	HPF_Den2: LREAL;
	ppsimbar: LREAL;
	prsimbar: LREAL;
END_VAR
VAR_OUTPUT
	uPF: LREAL;
END_VAR
VAR
	HP_Filter_tmp: LREAL;
	VectorConcatenate: ARRAY[0..1] OF LREAL;
	VectorConcatenate1: ARRAY[0..1] OF LREAL;
	HP_Filter_states: LREAL;
END_VAR



CASE ssMethodType OF
    0: 
        (* InitializeConditions for DiscreteTransferFcn: '<S1>/HP_Filter' *)
        HP_Filter_states := 0.0;
    1: 
        (* SignalConversion: '<S1>/ConcatBufferAtVector ConcatenateIn1' *)
        VectorConcatenate[0] := HPF_Num1;
        (* SignalConversion: '<S1>/ConcatBufferAtVector ConcatenateIn2' *)
        VectorConcatenate[1] := HPF_Num2;
        (* SignalConversion: '<S1>/ConcatBufferAtVector Concatenate1In1' *)
        VectorConcatenate1[0] := HPF_Den1;
        (* SignalConversion: '<S1>/ConcatBufferAtVector Concatenate1In2' *)
        VectorConcatenate1[1] := HPF_Den2;
        (* DiscreteTransferFcn: '<S1>/HP_Filter' incorporates:
         *  Gain: '<S1>/Gain'
         *  Gain: '<S1>/Gain3'
         *  Gain: '<S1>/muC'
         *  Sum: '<S1>/Add' *)
        HP_Filter_tmp := ((100000.0 * ppsimbar) - ((100000.0 * prsimbar) * 0.7101)) - (VectorConcatenate1[1] * HP_Filter_states);
        (* Switch: '<S1>/Switch2' incorporates:
         *  Constant: '<S1>/Constant' *)

        IF Enable THEN 
            (* Switch: '<S1>/Switch1' incorporates:
             *  Constant: '<S1>/Constant'
             *  DiscreteTransferFcn: '<S1>/HP_Filter'
             *  Product: '<S1>/Product' *)

            IF usDelay > 2.0 THEN 
                uPF := ((VectorConcatenate[0] * HP_Filter_tmp) + (VectorConcatenate[1] * HP_Filter_states)) * kQf;
            ELSE 
                uPF := 0.0;
            END_IF;

            (* End of Switch: '<S1>/Switch1' *)
        ELSE 
            uPF := 0.0;
        END_IF;

        (* End of Switch: '<S1>/Switch2' *)
        

        (* Saturate: '<S1>/Saturation5' *)

        IF uPF >= 3600.0 THEN 
            uPF := 3600.0;
        ELSIF uPF <= -3600.0 THEN 
            uPF := -3600.0;
        END_IF;

        (* End of Saturate: '<S1>/Saturation5' *)
        

        (* Update for DiscreteTransferFcn: '<S1>/HP_Filter' *)
        HP_Filter_states := HP_Filter_tmp;
END_CASE;

END_FUNCTION_BLOCK

// IndraMotionMlc1/Application/SCC_Controller_PFB
FUNCTION_BLOCK SCC_Controller_PFB
VAR_INPUT
	ssMethodType: SINT;
	FB_Cntr_On: BOOL;
	I_Cntr_On: BOOL;
	k_P: LREAL;
	k_I: LREAL;
	xC_Ref: LREAL;
	xC: LREAL;
	Clock: LREAL;
END_VAR
VAR_OUTPUT
	u_P: LREAL;
	u_I: LREAL;
	I_reset: LREAL;
	Pos_Error: LREAL;
	u_FB: LREAL;
END_VAR
VAR
	rtb_Sum1: LREAL;
	rtb_u_FB: LREAL;
	c_DiscreteTimeIntegrator_DS: LREAL;
END_VAR



CASE ssMethodType OF
    0: 
        (* InitializeConditions for DiscreteIntegrator: '<S1>/Discrete-Time Integrator' *)
        c_DiscreteTimeIntegrator_DS := 0.0;
    1: 
        (* MATLAB Function: '<S1>/Controller_Reset' *)
        (* MATLAB Function 'SCC_Controller_PFB/Controller_Reset': '<S2>:1' *)
        (* '<S2>:1:3' I_Reset = 1; *)
        (* '<S2>:1:5' if Clock > 0 *)

        IF Clock > 0.0 THEN 
            (* '<S2>:1:6' I_Reset = 0; *)
            I_reset := 0.0;
        ELSE 
            (* '<S2>:1:7' else *)
            (* '<S2>:1:8' I_Reset = 1; *)
            I_reset := 1.0;
            (* DiscreteIntegrator: '<S1>/Discrete-Time Integrator' *)
            c_DiscreteTimeIntegrator_DS := 0.0;
        END_IF;

        (* End of MATLAB Function: '<S1>/Controller_Reset' *)
        

        (* Sum: '<S1>/Sum1' incorporates:
         *  Gain: '<S1>/Gain1'
         *  Gain: '<S1>/Gain2' *)
        rtb_Sum1 := (0.001 * xC_Ref) - (0.001 * xC);
        (* Product: '<S1>/Product' *)
        u_P := k_P * rtb_Sum1;
        (* Switch: '<S1>/Switch' incorporates:
         *  Constant: '<S1>/Constant'
         *  DiscreteIntegrator: '<S1>/Discrete-Time Integrator' *)

        IF I_Cntr_On THEN 
            u_I := c_DiscreteTimeIntegrator_DS;
        ELSE 
            u_I := 0.0;
        END_IF;

        (* End of Switch: '<S1>/Switch' *)
        

        (* Sum: '<S1>/Sum5' *)
        rtb_u_FB := u_P + u_I;
        (* Saturate: '<S1>/Saturation1' *)

        IF rtb_u_FB >= 376.99111843077515 THEN 
            u_FB := 376.99111843077515;
        ELSIF rtb_u_FB > -376.99111843077515 THEN 
            u_FB := rtb_u_FB;
        ELSE 
            u_FB := -376.99111843077515;
        END_IF;

        (* End of Saturate: '<S1>/Saturation1' *)
        

        (* Sum: '<S1>/Sum3' *)
        rtb_u_FB := u_FB - rtb_u_FB;
        (* Switch: '<S1>/Switch1' incorporates:
         *  Constant: '<S1>/Constant1' *)

        IF  NOT FB_Cntr_On THEN 
            u_FB := 0.0;
        END_IF;

        (* End of Switch: '<S1>/Switch1' *)
        

        (* Gain: '<S1>/Gain' *)
        u_FB := 9.5492965855137211 * u_FB;
        (* Outport: '<Root>/Pos_Error' incorporates:
         *  Gain: '<S1>/Gain3' *)
        Pos_Error := 1000.0 * rtb_Sum1;
        (* Update for DiscreteIntegrator: '<S1>/Discrete-Time Integrator' incorporates:
         *  Product: '<S1>/Divide'
         *  Product: '<S1>/Product2'
         *  Sum: '<S1>/Sum2' *)
        c_DiscreteTimeIntegrator_DS := ((((rtb_u_FB / k_P) + rtb_Sum1) * k_I) * 0.001) + c_DiscreteTimeIntegrator_DS;
END_CASE;

END_FUNCTION_BLOCK

// IndraMotionMlc1/Application/SCC_Controller_VFF
FUNCTION_BLOCK SCC_Controller_VFF
VAR_INPUT
	Enable: BOOL;
	kq_Up: LREAL;
	kq_Down: LREAL;
	vC_Ref: LREAL;
END_VAR
VAR_OUTPUT
	u_FF: LREAL;
END_VAR
VAR
	rtb_Switch1: LREAL;
END_VAR


(* Gain: '<S1>/Gain3' incorporates:
 *  Gain: '<S1>/Gain1' *)
rtb_Switch1 := (0.001 * vC_Ref) * 0.0033183072403542195;
(* Switch: '<S1>/Switch' *)

IF rtb_Switch1 >= 0.0 THEN 
    (* Outport: '<Root>/u_FF' incorporates:
     *  Product: '<S1>/Divide1' *)
    u_FF := rtb_Switch1 / kq_Up;
ELSE 
    (* Outport: '<Root>/u_FF' incorporates:
     *  Product: '<S1>/Divide2' *)
    u_FF := rtb_Switch1 / kq_Down;
END_IF;

(* End of Switch: '<S1>/Switch' *)


(* Switch: '<S1>/Switch1' *)

IF  NOT Enable THEN 
    (* Outport: '<Root>/u_FF' incorporates:
     *  Constant: '<S1>/Constant' *)
    u_FF := 0.0;
END_IF;

(* End of Switch: '<S1>/Switch1' *)

END_FUNCTION_BLOCK

// IndraMotionMlc1/Application/SCC_PFB_Controller_PID
FUNCTION_BLOCK SCC_PFB_Controller_PID
VAR_INPUT
	ssMethodType: SINT;
	FB_Cntr_On: BOOL;
	I_Cntr_On: BOOL;
	k_P: LREAL;
	k_I: LREAL;
	xC_Ref: LREAL;
	xC: LREAL;
	Clock: LREAL;
	D_Cntr_On: BOOL;
	Lead_Num1: LREAL;
	Lead_Num2: LREAL;
	Lead_Den1: LREAL;
	Lead_Den2: LREAL;
END_VAR
VAR_OUTPUT
	u_P: LREAL;
	u_I: LREAL;
	I_reset: LREAL;
	Pos_Error: LREAL;
	u_FB: LREAL;
END_VAR
VAR
	rtb_Sum1: LREAL;
	rtb_u_FB: LREAL;
	rtb_Sum5: LREAL;
	DiscreteTransferFcn_tmp: LREAL;
	c_DiscreteTimeIntegrator_DS: LREAL;
	VectorConcatenate: ARRAY[0..1] OF LREAL;
	VectorConcatenate1: ARRAY[0..1] OF LREAL;
	DiscreteTransferFcn_states: LREAL;
END_VAR



CASE ssMethodType OF
    0: 
        (* InitializeConditions for DiscreteIntegrator: '<S1>/Discrete-Time Integrator' *)
        c_DiscreteTimeIntegrator_DS := 0.0;
        (* InitializeConditions for DiscreteTransferFcn: '<S1>/Discrete Transfer Fcn' *)
        DiscreteTransferFcn_states := 0.0;
    1: 
        (* MATLAB Function: '<S1>/Controller_Reset' *)
        (* MATLAB Function 'SCC_PFB_Controller_PID/Controller_Reset': '<S2>:1' *)
        (* '<S2>:1:3' I_Reset = 1; *)
        (* '<S2>:1:5' if Clock > 0 *)

        IF Clock > 0.0 THEN 
            (* '<S2>:1:6' I_Reset = 0; *)
            I_reset := 0.0;
        ELSE 
            (* '<S2>:1:7' else *)
            (* '<S2>:1:8' I_Reset = 1; *)
            I_reset := 1.0;
        END_IF;

        (* End of MATLAB Function: '<S1>/Controller_Reset' *)
        

        (* Sum: '<S1>/Sum1' incorporates:
         *  Gain: '<S1>/Gain1'
         *  Gain: '<S1>/Gain2' *)
        rtb_Sum1 := (0.001 * xC_Ref) - (0.001 * xC);
        (* Product: '<S1>/Product' *)
        u_P := k_P * rtb_Sum1;
        (* DiscreteIntegrator: '<S1>/Discrete-Time Integrator' *)

        IF I_reset <> 0.0 THEN 
            c_DiscreteTimeIntegrator_DS := 0.0;
        END_IF;

        (* Switch: '<S1>/Switch' incorporates:
         *  Constant: '<S1>/Constant'
         *  DiscreteIntegrator: '<S1>/Discrete-Time Integrator' *)

        IF I_Cntr_On THEN 
            u_I := c_DiscreteTimeIntegrator_DS;
        ELSE 
            u_I := 0.0;
        END_IF;

        (* End of Switch: '<S1>/Switch' *)
        

        (* Sum: '<S1>/Sum5' *)
        rtb_Sum5 := u_P + u_I;
        (* SignalConversion: '<S1>/ConcatBufferAtVector ConcatenateIn1' *)
        VectorConcatenate[0] := Lead_Num1;
        (* SignalConversion: '<S1>/ConcatBufferAtVector ConcatenateIn2' *)
        VectorConcatenate[1] := Lead_Num2;
        (* SignalConversion: '<S1>/ConcatBufferAtVector Concatenate1In1' *)
        VectorConcatenate1[0] := Lead_Den1;
        (* SignalConversion: '<S1>/ConcatBufferAtVector Concatenate1In2' *)
        VectorConcatenate1[1] := Lead_Den2;
        (* DiscreteTransferFcn: '<S1>/Discrete Transfer Fcn' *)
        DiscreteTransferFcn_tmp := rtb_Sum5 - (VectorConcatenate1[1] * DiscreteTransferFcn_states);
        rtb_u_FB := (VectorConcatenate[0] * DiscreteTransferFcn_tmp) + (VectorConcatenate[1] * DiscreteTransferFcn_states);
        (* Switch: '<S1>/Switch2' *)

        IF  NOT D_Cntr_On THEN 
            rtb_u_FB := rtb_Sum5;
        END_IF;

        (* End of Switch: '<S1>/Switch2' *)
        

        (* Saturate: '<S1>/Saturation1' *)

        IF rtb_u_FB >= 376.99111843077515 THEN 
            u_FB := 376.99111843077515;
        ELSIF rtb_u_FB > -376.99111843077515 THEN 
            u_FB := rtb_u_FB;
        ELSE 
            u_FB := -376.99111843077515;
        END_IF;

        (* End of Saturate: '<S1>/Saturation1' *)
        

        (* Sum: '<S1>/Sum3' *)
        rtb_u_FB := u_FB - rtb_u_FB;
        (* Switch: '<S1>/Switch1' incorporates:
         *  Constant: '<S1>/Constant1' *)

        IF  NOT FB_Cntr_On THEN 
            u_FB := 0.0;
        END_IF;

        (* End of Switch: '<S1>/Switch1' *)
        

        (* Gain: '<S1>/Gain' *)
        u_FB := 9.5492965855137211 * u_FB;
        (* Outport: '<Root>/Pos_Error' incorporates:
         *  Gain: '<S1>/Gain3' *)
        Pos_Error := 1000.0 * rtb_Sum1;
        (* Update for DiscreteIntegrator: '<S1>/Discrete-Time Integrator' incorporates:
         *  Product: '<S1>/Divide'
         *  Product: '<S1>/Product2'
         *  Sum: '<S1>/Sum2' *)
        c_DiscreteTimeIntegrator_DS := ((((rtb_u_FB / k_P) + rtb_Sum1) * k_I) * 0.001) + c_DiscreteTimeIntegrator_DS;
        (* Update for DiscreteTransferFcn: '<S1>/Discrete Transfer Fcn' *)
        DiscreteTransferFcn_states := DiscreteTransferFcn_tmp;
END_CASE;

END_FUNCTION_BLOCK

// IndraMotionMlc1/Application/SCC_PFB_Controller_PID2
FUNCTION_BLOCK SCC_PFB_Controller_PID2
VAR_INPUT
	ssMethodType: SINT;
	FB_Cntr_On: BOOL;
	I_Cntr_On: BOOL;
	k_P: LREAL;
	k_I: LREAL;
	xC_Ref: LREAL;
	xC: LREAL;
	Clock: LREAL;
	D_Cntr_On: BOOL;
	D_Num1: LREAL;
	D_Num2: LREAL;
	D_Den1: LREAL;
	D_Den2: LREAL;
	D_Den3: LREAL;
END_VAR
VAR_OUTPUT
	u_P: LREAL;
	u_I: LREAL;
	I_reset: LREAL;
	Pos_Error: LREAL;
	u_FB: LREAL;
END_VAR
VAR
	denAccum: LREAL;
	rtb_u_FB: LREAL;
	Sum1: LREAL;
	VectorConcatenate: ARRAY[0..1] OF LREAL;
	VectorConcatenate1: ARRAY[0..2] OF LREAL;
	c_DiscreteTimeIntegrator_DS: LREAL;
	DiscreteTransferFcn_states: ARRAY[0..1] OF LREAL;
END_VAR



CASE ssMethodType OF
    0: 
        (* InitializeConditions for DiscreteTransferFcn: '<S1>/Discrete Transfer Fcn' *)
        DiscreteTransferFcn_states[0] := 0.0;
        DiscreteTransferFcn_states[1] := 0.0;
        (* InitializeConditions for DiscreteIntegrator: '<S1>/Discrete-Time Integrator' *)
        c_DiscreteTimeIntegrator_DS := 0.0;
    1: 
        (* MATLAB Function: '<S1>/Controller_Reset' *)
        (* MATLAB Function 'SCC_PFB_Controller_PID2/Controller_Reset': '<S2>:1' *)
        (* '<S2>:1:3' I_Reset = 1; *)
        (* '<S2>:1:5' if Clock > 0 *)

        IF Clock > 0.0 THEN 
            (* '<S2>:1:6' I_Reset = 0; *)
            I_reset := 0.0;
        ELSE 
            (* '<S2>:1:7' else *)
            (* '<S2>:1:8' I_Reset = 1; *)
            I_reset := 1.0;
        END_IF;

        (* End of MATLAB Function: '<S1>/Controller_Reset' *)
        

        (* SignalConversion: '<S1>/ConcatBufferAtVector ConcatenateIn1' *)
        VectorConcatenate[0] := D_Num1;
        (* SignalConversion: '<S1>/ConcatBufferAtVector ConcatenateIn2' *)
        VectorConcatenate[1] := D_Num2;
        (* SignalConversion: '<S1>/ConcatBufferAtVector Concatenate1In1' *)
        VectorConcatenate1[0] := D_Den1;
        (* SignalConversion: '<S1>/ConcatBufferAtVector Concatenate1In2' *)
        VectorConcatenate1[1] := D_Den2;
        (* SignalConversion: '<S1>/ConcatBufferAtVector Concatenate1In3' *)
        VectorConcatenate1[2] := D_Den3;
        (* DiscreteTransferFcn: '<S1>/Discrete Transfer Fcn' *)
        rtb_u_FB := (VectorConcatenate[0] * DiscreteTransferFcn_states[0]) + (VectorConcatenate[1] * DiscreteTransferFcn_states[1]);
        (* DiscreteIntegrator: '<S1>/Discrete-Time Integrator' *)

        IF I_reset <> 0.0 THEN 
            c_DiscreteTimeIntegrator_DS := 0.0;
        END_IF;

        (* Sum: '<S1>/Sum1' incorporates:
         *  Gain: '<S1>/Gain1'
         *  Gain: '<S1>/Gain2' *)
        Sum1 := (0.001 * xC_Ref) - (0.001 * xC);
        (* Product: '<S1>/Product' *)
        u_P := k_P * Sum1;
        (* Switch: '<S1>/Switch' incorporates:
         *  Constant: '<S1>/Constant'
         *  DiscreteIntegrator: '<S1>/Discrete-Time Integrator' *)

        IF I_Cntr_On THEN 
            u_I := c_DiscreteTimeIntegrator_DS;
        ELSE 
            u_I := 0.0;
        END_IF;

        (* End of Switch: '<S1>/Switch' *)
        

        (* Switch: '<S1>/Switch2' incorporates:
         *  Constant: '<S1>/Constant2' *)

        IF  NOT D_Cntr_On THEN 
            rtb_u_FB := 0.0;
        END_IF;

        (* End of Switch: '<S1>/Switch2' *)
        

        (* Sum: '<S1>/Sum5' *)
        rtb_u_FB := (u_P + u_I) + rtb_u_FB;
        (* Saturate: '<S1>/Saturation1' *)

        IF rtb_u_FB >= 335.10321638291128 THEN 
            u_FB := 335.10321638291128;
        ELSIF rtb_u_FB > -335.10321638291128 THEN 
            u_FB := rtb_u_FB;
        ELSE 
            u_FB := -335.10321638291128;
        END_IF;

        (* End of Saturate: '<S1>/Saturation1' *)
        

        (* Sum: '<S1>/Sum3' *)
        rtb_u_FB := u_FB - rtb_u_FB;
        (* Switch: '<S1>/Switch1' incorporates:
         *  Constant: '<S1>/Constant1' *)

        IF  NOT FB_Cntr_On THEN 
            u_FB := 0.0;
        END_IF;

        (* End of Switch: '<S1>/Switch1' *)
        

        (* Gain: '<S1>/Gain' *)
        u_FB := 9.5492965855137211 * u_FB;
        (* Saturate: '<S1>/Saturation2' *)

        IF u_FB >= 3200.0 THEN 
            u_FB := 3200.0;
        ELSIF u_FB <= -3200.0 THEN 
            u_FB := -3200.0;
        END_IF;

        (* End of Saturate: '<S1>/Saturation2' *)
        

        (* Outport: '<Root>/Pos_Error' incorporates:
         *  Gain: '<S1>/Gain3' *)
        Pos_Error := 1000.0 * Sum1;
        (* Update for DiscreteTransferFcn: '<S1>/Discrete Transfer Fcn' *)
        denAccum := (Sum1 - (VectorConcatenate1[1] * DiscreteTransferFcn_states[0])) - (VectorConcatenate1[2] * DiscreteTransferFcn_states[1]);
        DiscreteTransferFcn_states[1] := DiscreteTransferFcn_states[0];
        DiscreteTransferFcn_states[0] := denAccum;
        (* Update for DiscreteIntegrator: '<S1>/Discrete-Time Integrator' incorporates:
         *  Product: '<S1>/Divide'
         *  Product: '<S1>/Product2'
         *  Sum: '<S1>/Sum2' *)
        c_DiscreteTimeIntegrator_DS := ((((rtb_u_FB / k_P) + Sum1) * k_I) * 0.001) + c_DiscreteTimeIntegrator_DS;
END_CASE;

END_FUNCTION_BLOCK

// IndraMotionMlc1/Application/SinuousCurve_Test
FUNCTION_BLOCK SinuousCurve_Test
VAR_INPUT
	Enable: BOOL;
	t0: LREAL;
	T_test: LREAL;
	x0: LREAL;
	Amp: LREAL;
	Freq: LREAL;
	CyclicTime: LREAL;
END_VAR
VAR_OUTPUT
	Valve_Opening_Ref: LREAL;
	T: LREAL;
END_VAR
VAR
END_VAR


(* MATLAB Function: '<S1>/WaveSignal' *)
(* MATLAB Function 'SinuousCurve_Test/WaveSignal': '<S2>:1' *)
(* '<S2>:1:3' if t>=t0 &amp;&amp; t<T_test *)

IF (CyclicTime >= t0) AND (CyclicTime < T_test) THEN 
    (* '<S2>:1:4' x = x0+A*sin(2*pi*f*(t-t0)); *)
    Valve_Opening_Ref := (SIN((6.2831853071795862 * Freq) * (CyclicTime - t0)) * Amp) + x0;
ELSE 
    (* '<S2>:1:5' else *)
    (* '<S2>:1:6' x = x0; *)
    Valve_Opening_Ref := x0;
END_IF;

(* Switch: '<S1>/Switch' *)
(* '<S2>:1:9' T = 1/f; *)

IF  NOT Enable THEN 
    (* Outport: '<Root>/Valve_Opening_Ref' *)
    Valve_Opening_Ref := x0;
END_IF;

(* End of Switch: '<S1>/Switch' *)


(* Outport: '<Root>/T' incorporates:
 *  MATLAB Function: '<S1>/WaveSignal' *)
T := 1.0 / Freq;

END_FUNCTION_BLOCK

// IndraMotionMlc1/Application/CascadedControllerFilter
FUNCTION_BLOCK CascadedControllerFilter
VAR_INPUT
	ssMethodType: SINT;
	Input: LREAL;
	HPF_Num1: LREAL;
	HPF_Num2: LREAL;
	HPF_Num3: LREAL;
	HPF_Den1: LREAL;
	HPF_Den2: LREAL;
	HPF_Den3: LREAL;
END_VAR
VAR_OUTPUT
	Output: LREAL;
END_VAR
VAR
	HP_Filter_tmp: LREAL;
	VectorConcatenate: ARRAY[0..2] OF LREAL;
	VectorConcatenate1: ARRAY[0..2] OF LREAL;
	HP_Filter_states: ARRAY[0..1] OF LREAL;
END_VAR



CASE ssMethodType OF
    0: 
        (* InitializeConditions for DiscreteTransferFcn: '<S1>/HP_Filter' *)
        HP_Filter_states[0] := 0.0;
        HP_Filter_states[1] := 0.0;
    1: 
        (* SignalConversion: '<S1>/ConcatBufferAtVector ConcatenateIn1' *)
        VectorConcatenate[0] := HPF_Num1;
        (* SignalConversion: '<S1>/ConcatBufferAtVector ConcatenateIn2' *)
        VectorConcatenate[1] := HPF_Num2;
        (* SignalConversion: '<S1>/ConcatBufferAtVector ConcatenateIn3' *)
        VectorConcatenate[2] := HPF_Num3;
        (* SignalConversion: '<S1>/ConcatBufferAtVector Concatenate1In1' *)
        VectorConcatenate1[0] := HPF_Den1;
        (* SignalConversion: '<S1>/ConcatBufferAtVector Concatenate1In2' *)
        VectorConcatenate1[1] := HPF_Den2;
        (* SignalConversion: '<S1>/ConcatBufferAtVector Concatenate1In3' *)
        VectorConcatenate1[2] := HPF_Den3;
        (* DiscreteTransferFcn: '<S1>/HP_Filter' *)
        HP_Filter_tmp := (Input - (VectorConcatenate1[1] * HP_Filter_states[0])) - (VectorConcatenate1[2] * HP_Filter_states[1]);
        (* Outport: '<Root>/Output' incorporates:
         *  DiscreteTransferFcn: '<S1>/HP_Filter' *)
        Output := ((VectorConcatenate[0] * HP_Filter_tmp) + (VectorConcatenate[1] * HP_Filter_states[0])) + (VectorConcatenate[2] * HP_Filter_states[1]);
        (* Update for DiscreteTransferFcn: '<S1>/HP_Filter' *)
        HP_Filter_states[1] := HP_Filter_states[0];
        HP_Filter_states[0] := HP_Filter_tmp;
END_CASE;

END_FUNCTION_BLOCK

// IndraMotionMlc1/Application/LHV_Controller
FUNCTION_BLOCK LHV_Controller
VAR_INPUT
	LHC_On: BOOL;
	SM_On: BOOL;
	v_set: LREAL;
	kP: LREAL;
	p_3: LREAL;
	p_1: LREAL;
END_VAR
VAR_OUTPUT
	error_bar: LREAL;
	Out_rpm: LREAL;
END_VAR
VAR
	rtb_u: LREAL;
	rtb_bar: BOOL;
END_VAR


(* Switch: '<S1>/Switch3' incorporates:
 *  Abs: '<S1>/Abs'
 *  Constant: '<S1>/Constant1' *)

IF ABS(v_set) > 0.0 THEN 
    rtb_bar := FALSE;
ELSE 
    rtb_bar := SM_On;
END_IF;

(* End of Switch: '<S1>/Switch3' *)


(* Switch: '<S1>/Switch6' incorporates:
 *  Constant: '<S1>/Constant7' *)

IF rtb_bar THEN 
    Out_rpm := p_1;
ELSE 
    Out_rpm := 0.0;
END_IF;

(* End of Switch: '<S1>/Switch6' *)


(* Gain: '<S1>/1' *)
rtb_u := 100000.0 * Out_rpm;
(* Switch: '<S1>/Switch5' incorporates:
 *  Constant: '<S1>/Constant7' *)

IF rtb_bar THEN 
    Out_rpm := p_3;
ELSE 
    Out_rpm := 0.0;
END_IF;

(* End of Switch: '<S1>/Switch5' *)


(* Sum: '<S1>/Add6' incorporates:
 *  Gain: '<S1>/12' *)
Out_rpm := (100000.0 * Out_rpm) - rtb_u;
(* Outport: '<Root>/error_bar' incorporates:
 *  Gain: '<S1>/Gain' *)
error_bar := 1.0E-5 * Out_rpm;
(* Switch: '<S1>/Switch1' incorporates:
 *  Constant: '<S1>/Constant'
 *  Gain: '<S1>/Gain15'
 *  Product: '<S1>/Product' *)

IF LHC_On THEN 
    Out_rpm := (Out_rpm * kP) * 9.5492965855137211;
ELSE 
    Out_rpm := 0.0;
END_IF;

(* End of Switch: '<S1>/Switch1' *)


(* Saturate: '<S1>/Saturation1' *)

IF Out_rpm >= 2000.0 THEN 
    Out_rpm := 2000.0;
ELSIF Out_rpm <= -2000.0 THEN 
    Out_rpm := -2000.0;
END_IF;

(* End of Saturate: '<S1>/Saturation1' *)

END_FUNCTION_BLOCK

// IndraMotionMlc1/Application/LHV_Enabler
FUNCTION_BLOCK LHV_Enabler
VAR_INPUT
	SM_ON: BOOL;
	LHC_error: LREAL;
	LHC_error_SP: LREAL;
END_VAR
VAR_OUTPUT
	LHV_Enable: LREAL;
END_VAR
VAR
END_VAR


(* MATLAB Function: '<S1>/MATLAB Function1' *)
(* MATLAB Function 'LHV_Enabler/MATLAB Function1': '<S2>:1' *)
(* '<S2>:1:4' if SM_ON > 0 &amp;&amp; abs(LHC_error)  < LHC_error_SP *)

IF SM_ON THEN 

    IF ABS(LHC_error) < LHC_error_SP THEN 
        (* Outport: '<Root>/LHV_Enable' *)
        (* '<S2>:1:5' y = 1; *)
        LHV_Enable := 1.0;
    ELSE 
        (* Outport: '<Root>/LHV_Enable' *)
        (* '<S2>:1:6' else *)
        (* '<S2>:1:7' y = 0; *)
        LHV_Enable := 0.0;
    END_IF;

ELSE 
    (* Outport: '<Root>/LHV_Enable' *)
    (* '<S2>:1:6' else *)
    (* '<S2>:1:7' y = 0; *)
    LHV_Enable := 0.0;
END_IF;

(* End of MATLAB Function: '<S1>/MATLAB Function1' *)

END_FUNCTION_BLOCK

// IndraMotionMlc1/Application/Pressure_Feed_Forward
FUNCTION_BLOCK Pressure_Feed_Forward
VAR_INPUT
	ssMethodType: SINT;
	SM_ON: BOOL;
	LHV_Enable: BOOL;
	p001: LREAL;
	p002: LREAL;
	v_ref: LREAL;
END_VAR
VAR_OUTPUT
	u_PFF: LREAL;
END_VAR
VAR
	tmp: LREAL;
	Subsystem2_Trig_ZCE: USINT;
	b_p001: LREAL;
END_VAR



CASE ssMethodType OF
    0: 
        (* SystemInitialize for Triggered SubSystem: '<S1>/Subsystem2' *)
        (* SystemInitialize for Outport: '<S3>/p001_Hold' *)
        b_p001 := 0.0;
        (* End of SystemInitialize for SubSystem: '<S1>/Subsystem2' *)
    1: 
        (* Outputs for Triggered SubSystem: '<S1>/Subsystem2' incorporates:
         *  TriggerPort: '<S3>/Trigger' *)

        IF ( NOT SM_ON) AND (Subsystem2_Trig_ZCE <> 0) THEN 
            (* Inport: '<S3>/p001' incorporates:
             *  Gain: '<S1>/Gain2' *)
            b_p001 := 100000.0 * p001;
        END_IF;

        Subsystem2_Trig_ZCE := BOOL_TO_USINT(SM_ON);
        (* End of Outputs for SubSystem: '<S1>/Subsystem2' *)
        

        (* MATLAB Function: '<S1>/MATLAB Function1' incorporates:
         *  Gain: '<S1>/Gain8' *)
        (* MATLAB Function 'Pressure_Feed_Forward/MATLAB Function1': '<S2>:1' *)
        (* '<S2>:1:3' if (p001_Hold - p_32) <= 0 *)
        tmp := b_p001 - (100000.0 * p002);

        IF tmp <= 0.0 THEN 
            (* '<S2>:1:4' FeedBackPressureTerm = 0; *)
            u_PFF := 0.0;
        ELSIF ABS(v_ref) > 0.0003 THEN 
            (* '<S2>:1:5' elseif abs(x_dot_ref) > 0.0003 *)
            (* '<S2>:1:6' FeedBackPressureTerm = 0; *)
            u_PFF := 0.0;
        ELSE 
            (* '<S2>:1:7' else *)
            (* '<S2>:1:8' FeedBackPressureTerm =  6.0256*10^(-5)/2 * (p001_Hold - p_32); *)
            u_PFF := tmp * 3.0127999999999997E-5;
        END_IF;

        (* End of MATLAB Function: '<S1>/MATLAB Function1' *)
        

        (* Switch: '<S1>/Switch' *)

        IF  NOT LHV_Enable THEN 
            (* Outport: '<Root>/u_PFF' incorporates:
             *  Constant: '<S1>/Constant' *)
            u_PFF := 0.0;
        END_IF;

        (* End of Switch: '<S1>/Switch' *)
END_CASE;

END_FUNCTION_BLOCK

// IndraMotionMlc1/Application/SCC_Primary_Controller
FUNCTION_BLOCK SCC_Primary_Controller
VAR_INPUT
	Enable: BOOL;
END_VAR
VAR_OUTPUT
	n_ref: REAL;
END_VAR
VAR
	Primary_Control3_0: Primary_Control3;
END_VAR
VAR // added by the converter: edge detectors and wires of the graphical bodies
    _w1 : BOOL;
END_VAR

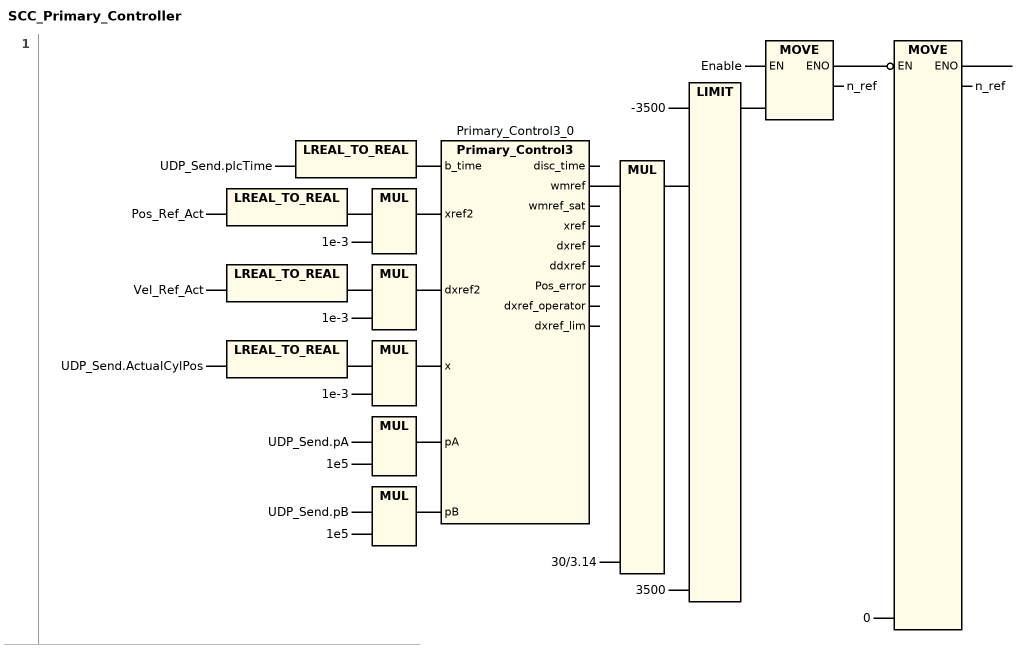
// NETWORK 1
Primary_Control3_0(
    b_time := LREAL_TO_REAL(UDP_Send.plcTime),
    xref2 := LREAL_TO_REAL(Pos_Ref_Act) * (1e-3),
    dxref2 := LREAL_TO_REAL(Vel_Ref_Act) * (1e-3),
    x := LREAL_TO_REAL(UDP_Send.ActualCylPos) * (1e-3),
    pA := UDP_Send.pA * 1e5,
    pB := UDP_Send.pB * 1e5); // Primary_Control3
_w1 := Enable;
IF _w1 THEN n_ref := LIMIT(-3500, Primary_Control3_0.wmref * (30/3.14), 3500); END_IF
IF NOT _w1 THEN n_ref := 0; END_IF

END_FUNCTION_BLOCK

// IndraMotionMlc1/Application/Primary_Control3
FUNCTION_BLOCK Primary_Control3
VAR_INPUT
	b_time: REAL;
	xref2: REAL;
	dxref2: REAL;
	x: REAL;
	pA: REAL;
	pB: REAL;
END_VAR
VAR_OUTPUT
	disc_time: REAL;
	wmref: REAL;
	wmref_sat: REAL;
	xref: REAL;
	dxref: REAL;
	ddxref: REAL;
	Pos_error: REAL;
	dxref_operator: REAL;
	dxref_lim: REAL;
END_VAR
VAR
	rate: REAL;
	e: REAL;
	uHP: REAL;
	ui: REAL;
	ei: REAL;
	uiold_not_empty: BOOL;
	eiold: REAL;
	dxref_lim_old: REAL;
	xref_old: REAL;
	wmref_sat_old: REAL;
	ddxref_old: REAL;
	ddxref_oldold: REAL;
	dxref_lim_oldold: REAL;
	dxref_old: REAL;
	dxref_oldold: REAL;
	wmref_old: REAL;
	pLold: REAL;
	uHPold: REAL;
	uiold: REAL;
	wm_ini: REAL := 0.62103355053102638;
	x_ini: REAL := 0.05;
	pA_ini: REAL := 6.9337754512426769E+6;
	A_B: REAL := 0.0023561944901923449;
	A_A: REAL := 0.0033183072403542195;
	pB_ini: REAL := 80830.0;
	Txm22: REAL := 0.001;
	slew_limit_ref: REAL := 0.10447093700391079;
	w_input: REAL := 6.2831853071795862;
	wad: REAL := 18.849555921538759;
	Cawx: REAL := 16.666666666666664;
	Cix: REAL := 3141.5926535897929;
	Cff: REAL := 2004.7633939712759;
	Cpx: REAL := 942.47779607693792;
	Cad: REAL := 5.2359877559829886E-6;
	wm_lim: REAL := 376.99111843077515;
	need_init: BOOL := TRUE;
END_VAR



IF need_init THEN 
    (* SystemInitialize for MATLAB Function: '<Root>/Primary_Control3' *)
    uiold_not_empty := FALSE;
    uiold := 0.0;
    dxref_lim_old := 0.0;
    dxref_lim_oldold := 0.0;
    dxref_old := 0.0;
    dxref_oldold := 0.0;
    ddxref_old := 0.0;
    ddxref_oldold := 0.0;
    uHPold := 0.0;
    need_init := FALSE;
END_IF;

(* MATLAB Function: '<Root>/Primary_Control3' *)
(* Motion controller (primary control) for SHA-type drive - Lasse Schmidt, ET/AAU - Date: 11-11-2020 *)
(* MATLAB Function 'Primary_Control3': '<S1>:1' *)
(* '<S1>:1:4' disc_time = time; *)
(* Sample time for control device *)
(* '<S1>:1:6' T=Txm22; *)
(* Initialization of variables *)

(* '<S1>:1:10' if isempty(uiold) *)

IF  NOT uiold_not_empty THEN 
    (* '<S1>:1:11' uiold = 0; *)
    uiold_not_empty := TRUE;
    (* '<S1>:1:12' eiold = wm_ini; *)
    eiold := wm_ini;
    (* '<S1>:1:13' dxref_lim_old = 0; *)
    (* '<S1>:1:14' dxref_lim_oldold = 0; *)
    (* '<S1>:1:15' dxref_old = 0; *)
    (* '<S1>:1:16' dxref_oldold = 0; *)
    (* '<S1>:1:17' ddxref_old = 0; *)
    (* '<S1>:1:18' ddxref_oldold = 0; *)
    (* '<S1>:1:19' xref_old = x_ini; *)
    xref_old := x_ini;
    (* '<S1>:1:20' wmref_sat_old = wm_ini; *)
    wmref_sat_old := wm_ini;
    (* '<S1>:1:21' wmref_old = wm_ini; *)
    wmref_old := wm_ini;
    (* '<S1>:1:22' pLold = (pA_ini-A_B/A_A*pB_ini); *)
    pLold := pA_ini - ((A_B / A_A) * pB_ini);
    (* '<S1>:1:23' uHPold = 0; *)
END_IF;

(* Reference generation *)
(* "Operator input" *)
(* '<S1>:1:27' k = 150/80; *)

(* '<S1>:1:28' dxref_operator = (time>=0)*(time<5/k)*0 + (time>=5/k)*(time<2*5/k)*80*k/1000 + (time>=2*5/k)*(time<4*5/k)*0 - (time>=4*5/k)*(time<5*5/k)*80*k/1000; *)
dxref_operator := (((DINT_TO_REAL(BOOL_TO_DINT(b_time >= 2.6666666666666665) * BOOL_TO_DINT(b_time < 5.333333333333333)) * 80.0) * 1.875) / 1000.0) - (((DINT_TO_REAL(BOOL_TO_DINT(b_time >= 10.666666666666666) * BOOL_TO_DINT(b_time < 13.333333333333334)) * 80.0) * 1.875) / 1000.0);
(* Rate limiter for of operator input *)
(* '<S1>:1:30' rate = (dxref_operator-dxref_lim_old)/Txm22; *)
rate := (dxref_operator - dxref_lim_old) / Txm22;
(* Limited rate of operator input *)
(* '<S1>:1:32' if abs(rate)<=slew_limit_ref *)

IF ABS(rate) > slew_limit_ref THEN 
    (* '<S1>:1:34' else *)
    (* '<S1>:1:35' F = slew_limit_ref*sign(rate); *)

    IF rate < 0.0 THEN 
        rate := -1.0;
    ELSIF rate > 0.0 THEN 
        rate := 1.0;
    END_IF;

    rate := slew_limit_ref * rate;
END_IF;

(* Limited "Operator input" *)
(* '<S1>:1:38' dxref_lim = F*T+dxref_lim_old; *)
dxref_lim := (rate * Txm22) + dxref_lim_old;
(* Limited and filtered reference(s) *)
(* '<S1>:1:40' ddxref = -(2*T^2*w_input^2*ddxref_old+T^2*w_input^2*ddxref_oldold-2*T*w_input^2*dxref_lim+2*T*w_input^2*dxref_lim_oldold-4*T*w_input*ddxref_oldold-8*ddxref_old+4*ddxref_oldold)/(T*w_input+2)^2; *)
rate := (Txm22 * w_input) + 2.0;
uHP := Txm22 * Txm22;
ui := w_input * w_input;
e := (2.0 * Txm22) * ui;
ei := (uHP * 2.0) * ui;
uHP := uHP * ui;
ui := (4.0 * Txm22) * w_input;
ddxref := ( -(((((((ei * ddxref_old) + (uHP * ddxref_oldold)) - (e * dxref_lim)) + (e * dxref_lim_oldold)) - (ui * ddxref_oldold)) - (8.0 * ddxref_old)) + (4.0 * ddxref_oldold))) / (rate * rate);
(* '<S1>:1:41' dxref = (T^2*w_input^2*dxref_lim+2*T^2*w_input^2*dxref_lim_old-2*T^2*w_input^2*dxref_old-T^2*w_input^2*dxref_oldold+T^2*w_input^2*dxref_lim_oldold+4*T*w_input*dxref_oldold+8*dxref_old-4*dxref_oldold)/(T*w_input+2)^2; *)
dxref := ((((((((ei * dxref_lim_old) + (uHP * dxref_lim)) - (ei * dxref_old)) - (uHP * dxref_oldold)) + (uHP * dxref_lim_oldold)) + (ui * dxref_oldold)) + (8.0 * dxref_old)) - (4.0 * dxref_oldold)) / (rate * rate);
(* '<S1>:1:42' xref = T/2*(dxref+dxref_old)+xref_old; *)
xref := ((Txm22 / 2.0) * (dxref + dxref_old)) + xref_old;
(* Controller - discrete implementation by forward euler transform *)
(* States used in motion controller *)
(* '<S1>:1:45' pL = pA - A_B/A_A*pB; *)
rate := pA - ((A_B / A_A) * pB);
(* '<S1>:1:46' e = xref2-x; *)
e := xref2 - x;
(* Output of high-pass pressure filter *)
(* '<S1>:1:48' if time > 0 *)

IF b_time > 0.0 THEN 
    (* '<S1>:1:49' uHP = -(T*wad*uHPold-2*pL+2*pLold-2*uHPold)/(T*wad+2); *)
    uHP := Txm22 * wad;
    uHP := ( -((((uHP * uHPold) - (2.0 * rate)) + (2.0 * pLold)) - (2.0 * uHPold))) / (uHP + 2.0);
ELSE 
    (* '<S1>:1:50' else *)
    (* '<S1>:1:51' uHP = 0; *)
    uHP := 0.0;
END_IF;

(* Integral control part  *)
(* '<S1>:1:55' if abs(xref2) > 0 *)

IF b_time > 0.0 THEN 
    (* Input to integral control term *)
    (* '<S1>:1:57' ui = (e - Cawx*(wmref_old-wmref_sat_old))*Cix; *)
    ui := (e - ((wmref_old - wmref_sat_old) * Cawx)) * Cix;
    (* Output of integral term of PI controller with anti wind-up loop *)
    (* '<S1>:1:59' ei = T/2*(ui+uiold)+eiold; *)
    ei := ((Txm22 / 2.0) * (ui + uiold)) + eiold;
ELSE 
    (* '<S1>:1:60' else *)
    (* '<S1>:1:61' ui = 0; *)
    ui := 0.0;
    (* '<S1>:1:62' ei = 0; *)
    ei := 0.0;
END_IF;

(* E-motor speed reference *)
(* '<S1>:1:65' wmref = Cff*dxref + Cpx*e + ei - Cad*uHP; *)
wmref := (((Cff * dxref2) + (Cpx * e)) + ei) - (Cad * uHP);
(* Limited E-motor speed reference *)
(* '<S1>:1:67' if abs(wmref)<=wm_lim *)

IF ABS(wmref) <= wm_lim THEN 
    (* '<S1>:1:68' wmref_sat = wmref; *)
    wmref_sat := wmref;
ELSE 
    (* '<S1>:1:69' else *)
    (* '<S1>:1:70' wmref_sat = wm_lim*sign(wmref); *)

    IF wmref < 0.0 THEN 
        e := -1.0;
    ELSIF wmref > 0.0 THEN 
        e := 1.0;
    ELSE 
        e := wmref;
    END_IF;

    wmref_sat := wm_lim * e;
END_IF;

(* Delayed states *)
(* '<S1>:1:73' uHPold=uHP; *)
uHPold := uHP;
(* '<S1>:1:74' pLold=pL; *)
pLold := rate;
(* '<S1>:1:75' eiold=ei; *)
eiold := ei;
(* '<S1>:1:76' uiold=ui; *)
uiold := ui;
(* '<S1>:1:77' dxref_lim_oldold=dxref_lim_old; *)
dxref_lim_oldold := dxref_lim_old;
(* '<S1>:1:78' dxref_lim_old=dxref_lim; *)
dxref_lim_old := dxref_lim;
(* '<S1>:1:79' dxref_oldold=dxref_old; *)
dxref_oldold := dxref_old;
(* '<S1>:1:80' dxref_old=dxref; *)
dxref_old := dxref;
(* '<S1>:1:81' ddxref_oldold = ddxref_old; *)
ddxref_oldold := ddxref_old;
(* '<S1>:1:82' ddxref_old = ddxref; *)
ddxref_old := ddxref;
(* '<S1>:1:83' xref_old = xref; *)
xref_old := xref;
(* '<S1>:1:84' wmref_sat_old = wmref_sat; *)
wmref_sat_old := wmref_sat;
(* '<S1>:1:85' wmref_old = wmref; *)
wmref_old := wmref;
(* Outport: '<Root>/disc_time' incorporates:
 *  MATLAB Function: '<Root>/Primary_Control3' *)
(* Position error *)
(* '<S1>:1:87' Pos_error = xref-x; *)
(* End *)
disc_time := b_time;
(* Outport: '<Root>/Pos_error' incorporates:
 *  MATLAB Function: '<Root>/Primary_Control3' *)
Pos_error := xref2 - x;

END_FUNCTION_BLOCK

// IndraMotionMlc1/Application/SCC_Secondary_Controller
FUNCTION_BLOCK SCC_Secondary_Controller
VAR_INPUT
	Enable: BOOL;
END_VAR
VAR_OUTPUT
	tau_ref: REAL;
END_VAR
VAR
	Secondary_Control_1: Secondary_Control;
	SC_constrol_status: BOOL :=FALSE;
	Kppx : REAL := 37.3999 ;
	Kix : REAL := 4.7872E+05 ;
    Kpx : REAL := 1.5929E+06 ;
	Kx : REAL := 3.3368 ;
//	Kawx : REAL := 0.0150 ;
	Kawx : REAL := 0.007;
	Low_Pass_Filter_0: Low_Pass_Filter;
	LPF_0: LPF;
	tLPF : REAL := 0.05; 
	LPF_1: LPF;
	Tmin: REAL := -80;
	Tmax: REAL := 80;
	LPF_2: LPF;
	LPF_3: LPF;
	LPF_4: LPF;
	error_mm: REAL;
	xref: REAL;
	dxref: REAL;
	ddxref: REAL;
	fLrefMan: REAL :=0;
	fLrefzero: REAL :=1;
	fLzero: REAL :=1;
	pA_zero: REAL :=1;
	pB_zero: REAL :=1;
	pA_man: REAL :=0;
	pB_man: REAL :=0;
END_VAR
VAR // added by the converter: edge detectors and wires of the graphical bodies
    _w1 : BOOL;
END_VAR

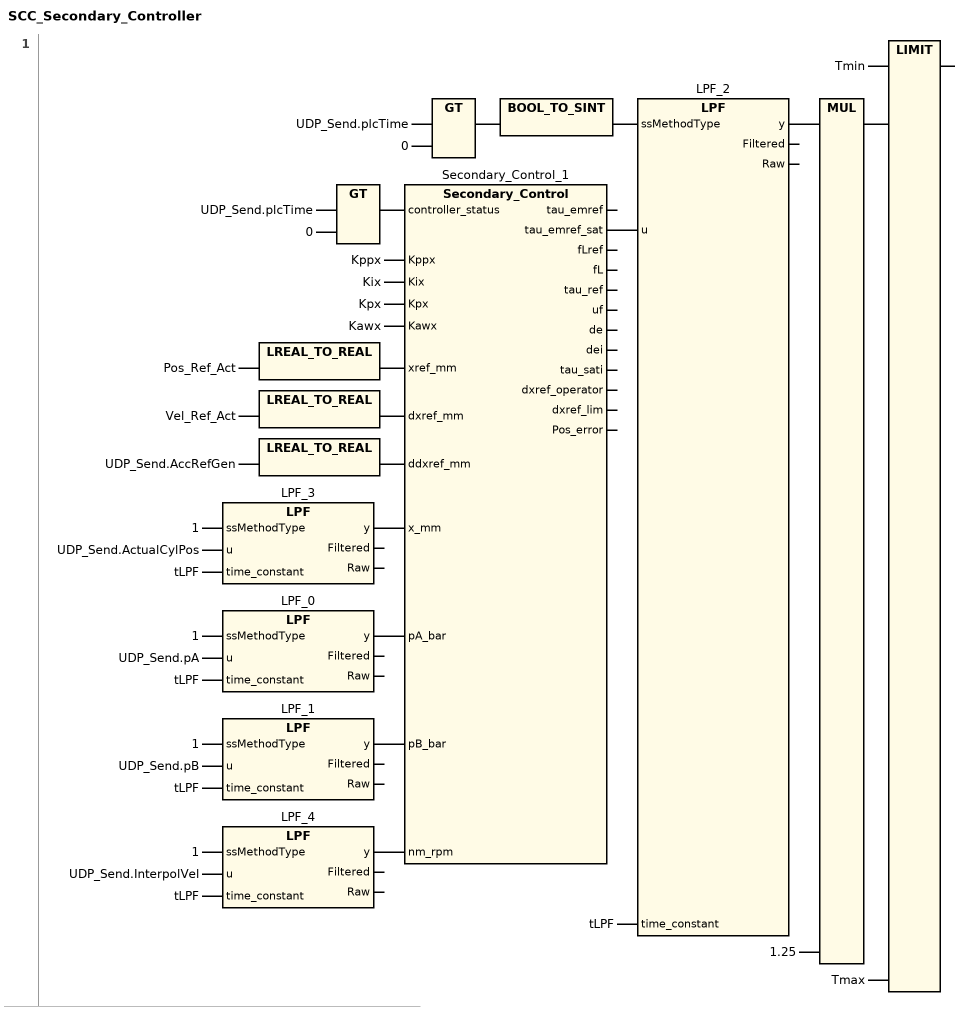
// NETWORK 1
LPF_3(ssMethodType := 1, u := UDP_Send.ActualCylPos, time_constant := tLPF); // LPF
LPF_0(ssMethodType := 1, u := UDP_Send.pA, time_constant := tLPF); // LPF
LPF_1(ssMethodType := 1, u := UDP_Send.pB, time_constant := tLPF); // LPF
LPF_4(ssMethodType := 1, u := UDP_Send.InterpolVel, time_constant := tLPF); // LPF
Secondary_Control_1(
    controller_status := UDP_Send.plcTime > 0,
    Kppx := Kppx,
    Kix := Kix,
    Kpx := Kpx,
    Kawx := Kawx,
    xref_mm := LREAL_TO_REAL(Pos_Ref_Act),
    dxref_mm := LREAL_TO_REAL(Vel_Ref_Act),
    ddxref_mm := LREAL_TO_REAL(UDP_Send.AccRefGen),
    x_mm := LPF_3.y,
    pA_bar := LPF_0.y,
    pB_bar := LPF_1.y,
    nm_rpm := LPF_4.y); // Secondary_Control
LPF_2(
    ssMethodType := BOOL_TO_SINT(UDP_Send.plcTime > 0),
    u := Secondary_Control_1.tau_emref_sat,
    time_constant := tLPF); // LPF
LIMIT(Tmin, LPF_2.y * 1.25, Tmax);

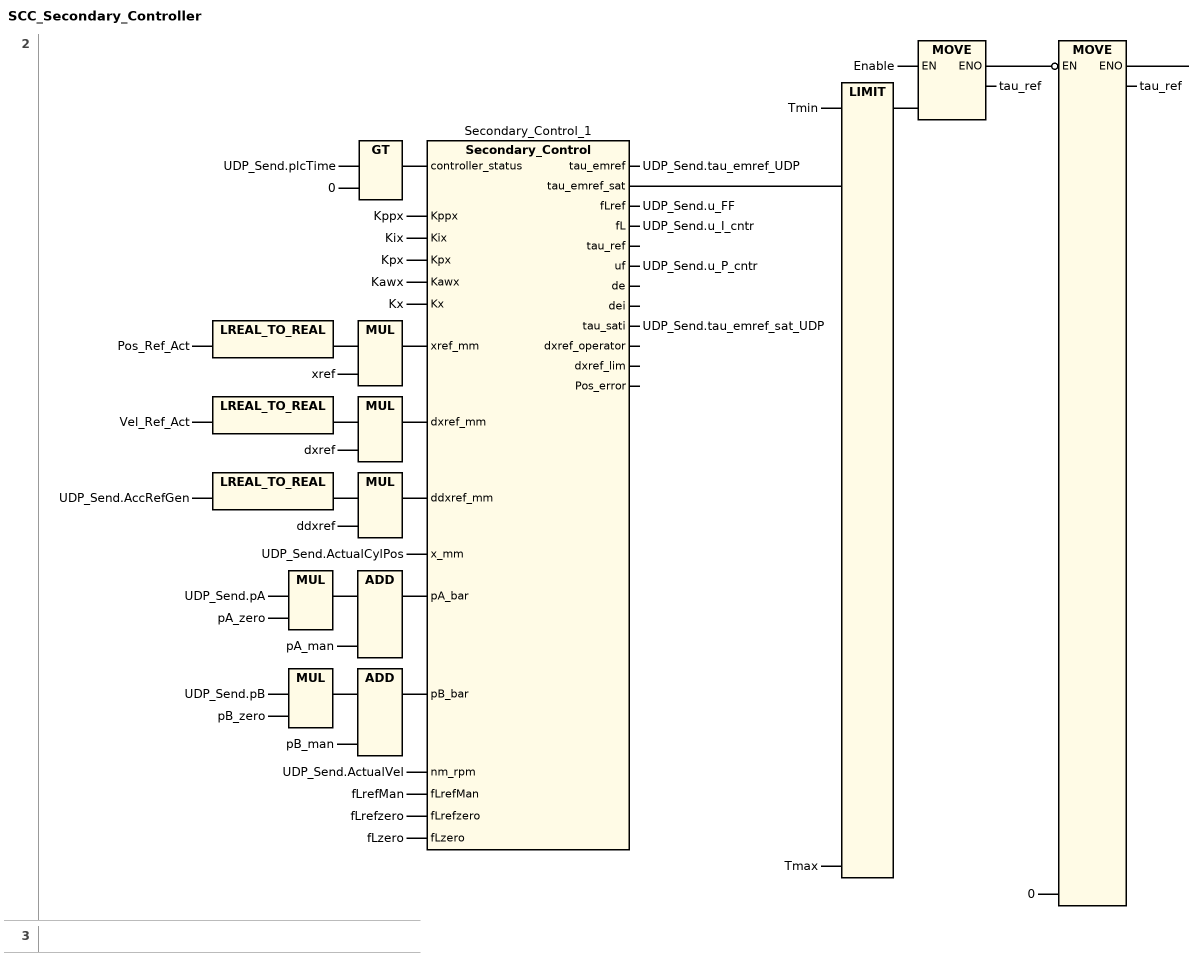
// NETWORK 2
Secondary_Control_1(
    controller_status := UDP_Send.plcTime > 0,
    Kppx := Kppx,
    Kix := Kix,
    Kpx := Kpx,
    Kawx := Kawx,
    Kx := Kx,
    xref_mm := LREAL_TO_REAL(Pos_Ref_Act) * xref,
    dxref_mm := LREAL_TO_REAL(Vel_Ref_Act) * dxref,
    ddxref_mm := LREAL_TO_REAL(UDP_Send.AccRefGen) * ddxref,
    x_mm := UDP_Send.ActualCylPos,
    pA_bar := UDP_Send.pA * pA_zero + pA_man,
    pB_bar := UDP_Send.pB * pB_zero + pB_man,
    nm_rpm := UDP_Send.ActualVel,
    fLrefMan := fLrefMan,
    fLrefzero := fLrefzero,
    fLzero := fLzero,
    tau_emref => UDP_Send.tau_emref_UDP,
    fLref => UDP_Send.u_FF,
    fL => UDP_Send.u_I_cntr,
    uf => UDP_Send.u_P_cntr,
    tau_sati => UDP_Send.tau_emref_sat_UDP); // Secondary_Control
_w1 := Enable;
IF _w1 THEN tau_ref := LIMIT(Tmin, Secondary_Control_1.tau_emref_sat, Tmax); END_IF
IF NOT _w1 THEN tau_ref := 0; END_IF

// NETWORK 3

END_FUNCTION_BLOCK

// IndraMotionMlc1/Application/LPF
FUNCTION_BLOCK LPF
VAR_INPUT
	ssMethodType: SINT;
	u: REAL;
	time_constant : REAL := 0.05;
END_VAR
VAR_OUTPUT
	y: REAL;
	Filtered: REAL;
	Raw: REAL;
END_VAR
VAR
	rtb_Compare: BOOL;
	Integrator_IC_LOADING: USINT;
	Integrator_PrevResetState: SINT;
	Integrator_DSTATE: REAL;
	Probe: ARRAY[0..1] OF REAL;
END_VAR



CASE ssMethodType OF
    0: 
        (* SystemInitialize for Atomic SubSystem: '<Root>/Low-Pass_Filter ' *)
        (* Start for Probe: '<S3>/Probe' *)
        Probe[0] := 0.001;
        Probe[1] := 0.0;
        (* InitializeConditions for DiscreteIntegrator: '<S8>/Integrator' *)
        Integrator_PrevResetState := 0;
        Integrator_IC_LOADING := 1;
        (* End of SystemInitialize for SubSystem: '<Root>/Low-Pass_Filter ' *)
    1: 
        (* Outputs for Atomic SubSystem: '<Root>/Low-Pass_Filter ' *)
        (* RelationalOperator: '<S6>/Compare' incorporates:
         *  Constant: '<S3>/Time constant'
         *  Constant: '<S6>/Constant'
         *  Sum: '<S3>/Sum1' *)
        rtb_Compare := (time_constant - Probe[0]) <= 0.0;
        (* DiscreteIntegrator: '<S8>/Integrator' *)

        IF Integrator_IC_LOADING <> 0 THEN 
            Integrator_DSTATE := u;
        END_IF;


        IF rtb_Compare OR (Integrator_PrevResetState <> 0) THEN 
            Integrator_DSTATE := u;
        END_IF;

        (* Outport: '<Root>/y' incorporates:
         *  DiscreteIntegrator: '<S8>/Integrator' *)
        y := Integrator_DSTATE;
        (* Update for DiscreteIntegrator: '<S8>/Integrator' incorporates:
         *  Constant: '<S3>/Time constant'
         *  MinMax: '<S3>/Max'
         *  Product: '<S2>/1//T'
         *  Sum: '<S2>/Sum1' *)
        Integrator_IC_LOADING := 0;
        Integrator_DSTATE := (((1.0 / MAX(Probe[0], time_constant)) * (u - Integrator_DSTATE)) * 0.001) + Integrator_DSTATE;

        IF rtb_Compare THEN 
            Integrator_PrevResetState := 1;
        ELSE 
            Integrator_PrevResetState := 0;
        END_IF;
      Filtered := y;
	  Raw := u;
		 
        (* End of Update for DiscreteIntegrator: '<S8>/Integrator' *)
        (* End of Outputs for SubSystem: '<Root>/Low-Pass_Filter ' *)
END_CASE;

END_FUNCTION_BLOCK

// IndraMotionMlc1/Application/Secondary_Control
FUNCTION_BLOCK Secondary_Control
VAR_INPUT
controller_status : BOOL ;	
Kppx : REAL;
Kix : REAL;
Kpx : REAL;
Kawx : REAL;
Kx : REAL;
xref_mm : REAL ;
dxref_mm : REAL ;
ddxref_mm : REAL ;

x_mm : REAL ;
pA_bar : REAL ;
pB_bar : REAL ;
nm_rpm : REAL ;
	fLrefMan: REAL;
	
	fLrefzero: REAL;
	fLzero: REAL;
	
END_VAR
VAR_OUTPUT
// Controller outputs
tau_emref : REAL ;
tau_emref_sat : REAL ;
fLref : REAL ;
fL : REAL ;
tau_ref : REAL ;
uf : REAL ;
de : REAL ;
dei : REAL ;
tau_sati : REAL ;
dxref_operator : REAL ;
dxref_lim : REAL ;

Pos_error : REAL ;
END_VAR
VAR
T : REAL := 1E-3 ;
// Reference variables
xref : REAL ;
dxref : REAL ;
ddxref : REAL ;


// Paramters

wL : REAL := 598.3986 ;
wh : REAL := 286.3657 ;
VAini : REAL := 0.0017 ;
VBini : REAL := 0.0022 ;
x_max : REAL := 0.5000 ;
betae : REAL := 600000000 ;
A_A : REAL := 0.0033 ;
A_B : REAL := 0.0024 ;
Jm : REAL := 0.0040 ;
Dpump : REAL := 1.6552E-06 ;
zetaL : REAL := 0.7071 ;

Ktau_max : REAL := 80 ;
slew_limit_ref : REAL := 0.1045 ;
w_input : REAL := 6.2832 ;

// control variables
x : REAL ;
pA : REAL ;
pB : REAL ;
wm : REAL ;

// i nitialisation variables
x_ini : REAL ;
Geq_ini : REAL ;
tau_emref_ini : REAL ;
controller_status_old : BOOL ;

// old values
x_old : REAL ;
xref_old : REAL ;
dxref_lim_old : REAL ;
dxref_lim_oldold : REAL ;
dxref_old : REAL ;
dxref_oldold : REAL ;
ddxref_old : REAL ;
ddxref_oldold : REAL ;
uf_old : REAL ;
de_old : REAL ;
dei_old : REAL ;
tau_emref_old : REAL ;
tau_emref_sat_old : REAL ;
tau_sati_old : REAL ;
tau_sat_old : REAL ;


tau_sat : REAL ;


VA : REAL ;
VB : REAL ;

END_VAR

 ///////////// Do input conversions here (from current/voltage signals tostates in SI units) ///////////////////////

x := x_mm*1E-3;
pA := pA_bar*1E5;  
pB := pB_bar*1E5;  
wm :=  nm_rpm*(3.14/30);
 
 ////////// initialisation of Controller/////////////////
Geq_ini := pA * A_A - pB * A_B ;
x_ini := x ;
tau_emref_ini := - ( A_A * x_ini + VAini ) * ( VBini + A_B * ( x_max - x_ini ) ) * wL* wL * ( A_A * pA - A_B * pB - Geq_ini ) * Jm / ( betae * Dpump * ( A_A * ( VBini + A_B * ( x_max - x_ini ) ) + A_B * ( A_A * x_ini + VAini ) ) ) + Dpump * ( pA - pB ) - Kx * wm ;

IF controller_status AND NOT ( controller_status_old ) THEN
x_old := x_ini;
xref_old := x_ini;
tau_emref_old := tau_emref_ini;
tau_emref_sat_old := tau_emref_ini;
END_IF

///////////////// Reference Generation////////////////////////

xref :=  xref_mm*1E-3;
dxref :=  dxref_mm*1E-3;
ddxref := ddxref_mm*1E-3;

///////////////// Control Algoritm////////////////////////
IF controller_status THEN
// Input TO piston velocity PI controller//
//Position P-controller and "piston velocity" feedback with first order low-pass filter
uf := ( ( Kppx * T * xref - Kppx * T * x - 2 * x ) * wh + ( Kppx * T * xref_old - Kppx * T * x_old + 2 * x_old ) * wh - ( T * wh - 2 ) * uf_old ) / ( T * wh + 2 ) ;
// "Piston velocity" control error (input to piston velocity PI-controller)
de := dxref + uf ;

// Controller - discrete implementation by bilinear transform (Tustin) //
//PI-controller integrator anti wind up loop
tau_sat := tau_emref_old - tau_emref_sat_old ;
tau_sati := T * Kawx * Kix / 2 * ( tau_sat + tau_sat_old ) + tau_sati_old ;
//Output of integral term of PI controller
dei := T * Kix / 2 * ( de + de_old ) + dei_old ;
//Piston force reference (PI-controller with integrator anti wind up)
fLref := (Kpx * de + dei - tau_sati)*fLrefzero + fLrefMan;

fL := (A_A * pA - A_B * pB)*fLzero ;
//Cylinder volumes
VA := VAini + A_A * x ;
VB := VBini + A_B * ( x_max - x ) ;
// Electro-magnetic torque reference
tau_ref := ( A_A * A_A * VB + A_B * A_B * VA ) * Jm * ( 2 * dxref * zetaL * wL + ddxref ) / ( Dpump * ( A_A * VB + A_B * VA ) ) - VA * VB * wL * wL * ( fL - fLref ) * Jm / ( betae * Dpump * ( A_A * VB + A_B * VA ) ) ;
tau_emref := tau_ref + Dpump * ( pA - pB ) - Kx * wm ;
// Limited electro-magnetic torque reference
IF ABS ( tau_emref ) <= Ktau_max THEN
tau_emref_sat := tau_emref ;
ELSE
tau_emref_sat := Ktau_max * ( tau_emref ) / ( ABS ( tau_emref ) ) ;
END_IF
ELSE
uf := 0 ;
de := 0 ;
tau_sat := 0 ;
tau_sati := 0 ;
dei := 0 ;
fLref := 0 ;
fL := 0 ;
tau_ref := 0 ;
tau_emref := 0 ;
tau_emref_sat := 0 ;
END_IF

/////////////////////// Assign old values///////////////////
tau_emref_old := tau_emref ;
tau_emref_sat_old := tau_emref_sat ;
tau_sati_old := tau_sati ;
tau_sat_old := tau_sat ;
de_old := de ;
dei_old := dei ;
uf_old := uf ;
x_old := x ;
dxref_lim_oldold := dxref_lim_old ;
dxref_lim_old := dxref_lim ;
dxref_oldold := dxref_old ;
dxref_old := dxref ;
ddxref_oldold := ddxref_old ;
ddxref_old := ddxref ;
xref_old := xref ;

controller_status_old := controller_status ;

// Position error
Pos_error := xref - x ;

END_FUNCTION_BLOCK

// IndraMotionMlc1/Application/Low_Pass_Filter
FUNCTION_BLOCK Low_Pass_Filter
VAR_INPUT
	In: LREAL;
	Num: LREAL;
	Den: LREAL;
END_VAR
VAR_OUTPUT
	Out: LREAL;
END_VAR
VAR
END_VAR


(* Outport: '<Root>/Out' incorporates:
 *  DiscreteTransferFcn: '<S1>/Discrete Transfer Fcn' *)
Out := In * Num;

END_FUNCTION_BLOCK

// IndraMotionMlc1/Application/CyclSercosChnl
FUNCTION_BLOCK CyclSercosChnl
VAR_INPUT
END_VAR
VAR_OUTPUT
	DataA: REAL; 
	DataB: REAL; 
	DataC: REAL; 
	DataD: REAL; 
	DataE: REAL; 
	DataF: REAL; 
END_VAR
VAR
END_VAR

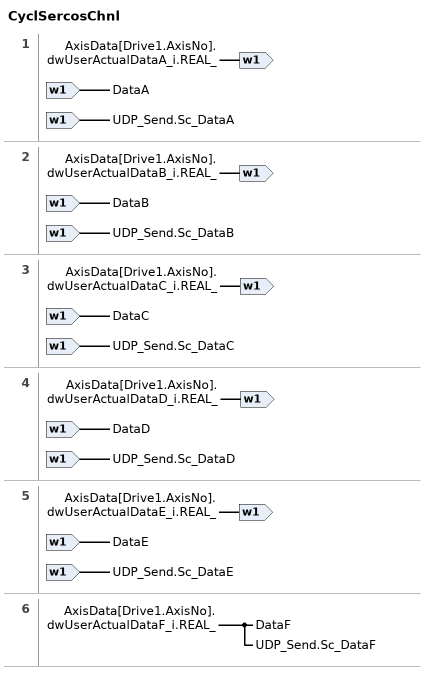
// NETWORK 1
DataA := AxisData[Drive1.AxisNo].dwUserActualDataA_i.REAL_;
UDP_Send.Sc_DataA := AxisData[Drive1.AxisNo].dwUserActualDataA_i.REAL_;

// NETWORK 2
DataB := AxisData[Drive1.AxisNo].dwUserActualDataB_i.REAL_;
UDP_Send.Sc_DataB := AxisData[Drive1.AxisNo].dwUserActualDataB_i.REAL_;

// NETWORK 3
DataC := AxisData[Drive1.AxisNo].dwUserActualDataC_i.REAL_;
UDP_Send.Sc_DataC := AxisData[Drive1.AxisNo].dwUserActualDataC_i.REAL_;

// NETWORK 4
DataD := AxisData[Drive1.AxisNo].dwUserActualDataD_i.REAL_;
UDP_Send.Sc_DataD := AxisData[Drive1.AxisNo].dwUserActualDataD_i.REAL_;

// NETWORK 5
DataE := AxisData[Drive1.AxisNo].dwUserActualDataE_i.REAL_;
UDP_Send.Sc_DataE := AxisData[Drive1.AxisNo].dwUserActualDataE_i.REAL_;

// NETWORK 6
DataF := AxisData[Drive1.AxisNo].dwUserActualDataF_i.REAL_;
UDP_Send.Sc_DataF := AxisData[Drive1.AxisNo].dwUserActualDataF_i.REAL_;

END_FUNCTION_BLOCK

// IndraMotionMlc1/Application/StepFunction_Test_Christian
FUNCTION_BLOCK StepFunction_Test_Christian
VAR_INPUT
	n_SP: LREAL;
	CyclicTime: LREAL;
	t0: LREAL;
	t1: LREAL;
	t2: LREAL;
	t3: LREAL;
	t4: LREAL;
	t5: LREAL;
	t6: LREAL;
	t7: LREAL;
	t8: LREAL;
	t9: LREAL;
	t10: LREAL;
	t11: LREAL;
	t12: LREAL;
	t13: LREAL;
END_VAR
VAR_OUTPUT
	n_ref: LREAL;
	EndTime: LREAL;
END_VAR
VAR
	tmp: LREAL;
	temp1: LREAL;
	temp2: LREAL;
END_VAR


(* MATLAB Function: '<S1>/StepFunction' *)
(* MATLAB Function 'StepFunction_Test_Christian/StepFunction': '<S2>:1' *)
(* '<S2>:1:2' if t==0 *)

IF CyclicTime = 0.0 THEN 
    (* Outport: '<Root>/n_ref' *)
    (* '<S2>:1:3' y = 0; *)
    n_ref := 0.0;
ELSIF (CyclicTime > 0.0) AND (CyclicTime < t0) THEN 
    (* Outport: '<Root>/n_ref' *)
    (* '<S2>:1:4' elseif t>0 &amp;&amp; t<t0 *)
    (* '<S2>:1:5' y = n_SP; *)
    n_ref := n_SP;
ELSE 
    tmp := t0 + t1;

    IF (CyclicTime >= t0) AND (CyclicTime < tmp) THEN 
        (* Outport: '<Root>/n_ref' *)
        (* '<S2>:1:6' elseif t>=(t0) &amp;&amp; t<(t0+t1) *)
        (* '<S2>:1:7' y = 0; *)
        n_ref := 0.0;
    ELSE 
        temp1 := tmp + t2;

        IF (CyclicTime >= tmp) AND (CyclicTime < temp1) THEN 
            (* Outport: '<Root>/n_ref' *)
            (* '<S2>:1:8' elseif t>=(t0+t1) &amp;&amp; t<(t0+t1+t2) *)
            (* '<S2>:1:9' y = n_SP; *)
            n_ref := n_SP;
        ELSE 
            tmp := temp1 + t3;

            IF (CyclicTime >= temp1) AND (CyclicTime < tmp) THEN 
                (* Outport: '<Root>/n_ref' *)
                (* '<S2>:1:10' elseif t>=(t0+t1+t2) &amp;&amp; t<(t0+t1+t2+t3) *)
                (* '<S2>:1:11' y = 0; *)
                n_ref := 0.0;
            ELSE 
                temp1 := tmp + t4;

                IF (CyclicTime >= tmp) AND (CyclicTime < temp1) THEN 
                    (* Outport: '<Root>/n_ref' *)
                    (* '<S2>:1:12' elseif t>=(t0+t1+t2+t3) &amp;&amp; t<(t0+t1+t2+t3+t4) *)
                    (* '<S2>:1:13' y = -n_SP; *)
                    n_ref :=  -n_SP;
                ELSE 
                    tmp := temp1 + t5;

                    IF (CyclicTime >= temp1) AND (CyclicTime < tmp) THEN 
                        (* Outport: '<Root>/n_ref' *)
                        (* '<S2>:1:14' elseif t>=(t0+t1+t2+t3+t4) &amp;&amp; t<(t0+t1+t2+t3+t4+t5) *)
                        (* '<S2>:1:15' y = 0; *)
                        n_ref := 0.0;
                    ELSE 
                        temp1 := tmp + t6;

                        IF (CyclicTime >= tmp) AND (CyclicTime < temp1) THEN 
                            (* Outport: '<Root>/n_ref' *)
                            (* '<S2>:1:16' elseif t>=(t0+t1+t2+t3+t4+t5) &amp;&amp; t<(t0+t1+t2+t3+t4+t5+t6) *)
                            (* '<S2>:1:17' y = n_SP; *)
                            n_ref := n_SP;
                        ELSE 
                            tmp := temp1 + t7;

                            IF (CyclicTime >= temp1) AND (CyclicTime < tmp) THEN 
                                (* Outport: '<Root>/n_ref' *)
                                (* '<S2>:1:18' elseif t>=(t0+t1+t2+t3+t4+t5+t6) &amp;&amp; t<(t0+t1+t2+t3+t4+t5+t6+t7) *)
                                (* '<S2>:1:19' y = -n_SP; *)
                                n_ref :=  -n_SP;
                            ELSE 
                                temp1 := tmp + t8;

                                IF (CyclicTime >= tmp) AND (CyclicTime < temp1) THEN 
                                    (* Outport: '<Root>/n_ref' *)
                                    (* '<S2>:1:20' elseif t>=(t0+t1+t2+t3+t4+t5+t6+t7) &amp;&amp; t<(t0+t1+t2+t3+t4+t5+t6+t7+t8) *)
                                    (* '<S2>:1:21' y = 0; *)
                                    n_ref := 0.0;
                                ELSE 
                                    tmp := temp1 + t9;

                                    IF (CyclicTime >= temp1) AND (CyclicTime < tmp) THEN 
                                        (* Outport: '<Root>/n_ref' *)
                                        (* '<S2>:1:22' elseif t>=(t0+t1+t2+t3+t4+t5+t6+t7+t8) &amp;&amp; t<(t0+t1+t2+t3+t4+t5+t6+t7+t8+t9) *)
                                        (* '<S2>:1:23' y = n_SP; *)
                                        n_ref := n_SP;
                                    ELSE 
                                        temp1 := tmp + t10;

                                        IF (CyclicTime >= tmp) AND (CyclicTime < temp1) THEN 
                                            (* Outport: '<Root>/n_ref' *)
                                            (* '<S2>:1:24' elseif t>=(t0+t1+t2+t3+t4+t5+t6+t7+t8+t9) &amp;&amp; t<(t0+t1+t2+t3+t4+t5+t6+t7+t8+t9+t10) *)
                                            (* '<S2>:1:25' y = 0; *)
                                            n_ref := 0.0;
                                        ELSE 
                                            tmp := temp1 + t11;

                                            IF (CyclicTime >= temp1) AND (CyclicTime < tmp) THEN 
                                                (* Outport: '<Root>/n_ref' *)
                                                (* '<S2>:1:26' elseif t>=(t0+t1+t2+t3+t4+t5+t6+t7+t8+t9+t10) &amp;&amp; t<(t0+t1+t2+t3+t4+t5+t6+t7+t8+t9+t10+t11) *)
                                                (* '<S2>:1:27' y = -n_SP; *)
                                                n_ref :=  -n_SP;
                                            ELSE 
                                                temp2 := tmp + t12;

                                                IF (CyclicTime >= tmp) AND (CyclicTime < temp2) THEN 
                                                    (* Outport: '<Root>/n_ref' *)
                                                    (* '<S2>:1:28' elseif t>=(t0+t1+t2+t3+t4+t5+t6+t7+t8+t9+t10+t11) &amp;&amp; t<(t0+t1+t2+t3+t4+t5+t6+t7+t8+t9+t10+t11+t12) *)
                                                    (* '<S2>:1:29' y = 0; *)
                                                    n_ref := 0.0;
                                                ELSE 
                                                    tmp := temp2 + t13;

                                                    IF (CyclicTime >= (temp1 + t12)) AND (CyclicTime < tmp) THEN 
                                                        (* Outport: '<Root>/n_ref' *)
                                                        (* '<S2>:1:30' elseif t>=(t0+t1+t2+t3+t4+t5+t6+t7+t8+t9+t10+t12) &amp;&amp; t<(t0+t1+t2+t3+t4+t5+t6+t7+t8+t9+t10+t11+t12+t13) *)
                                                        (* '<S2>:1:31' y = -n_SP; *)
                                                        n_ref :=  -n_SP;
                                                    ELSIF CyclicTime >= tmp THEN 
                                                        (* Outport: '<Root>/n_ref' *)
                                                        (* '<S2>:1:32' elseif t>=(t0+t1+t2+t3+t4+t5+t6+t7+t8+t9+t10+t11+t12+t13) *)
                                                        (* '<S2>:1:33' y = 0; *)
                                                        n_ref := 0.0;
                                                    ELSE 
                                                        (* Outport: '<Root>/n_ref' *)
                                                        (* '<S2>:1:34' else *)
                                                        (* '<S2>:1:35' y = 0; *)
                                                        n_ref := 0.0;
                                                    END_IF;

                                                END_IF;

                                            END_IF;

                                        END_IF;

                                    END_IF;

                                END_IF;

                            END_IF;

                        END_IF;

                    END_IF;

                END_IF;

            END_IF;

        END_IF;

    END_IF;

END_IF;

(* Outport: '<Root>/EndTime' incorporates:
 *  MATLAB Function: '<S1>/StepFunction' *)
(* '<S2>:1:38' T = t0+t1+t2+t3+t4+t5+t6+t7+t8+t9+t10+t11+t12; *)
EndTime := (((((((((((t0 + t1) + t2) + t3) + t4) + t5) + t6) + t7) + t8) + t9) + t10) + t11) + t12 + t13;

END_FUNCTION_BLOCK

// IndraMotionMlc1/Application/JoyStick_SCC_TrqCntrl
FUNCTION_BLOCK JoyStick_SCC_TrqCntrl
VAR_INPUT
	Enable: BOOL;
	Max_Torque: REAL;
	Init_Torqe: REAL;
END_VAR
VAR_OUTPUT
	JoyY_Ref: REAL;
END_VAR

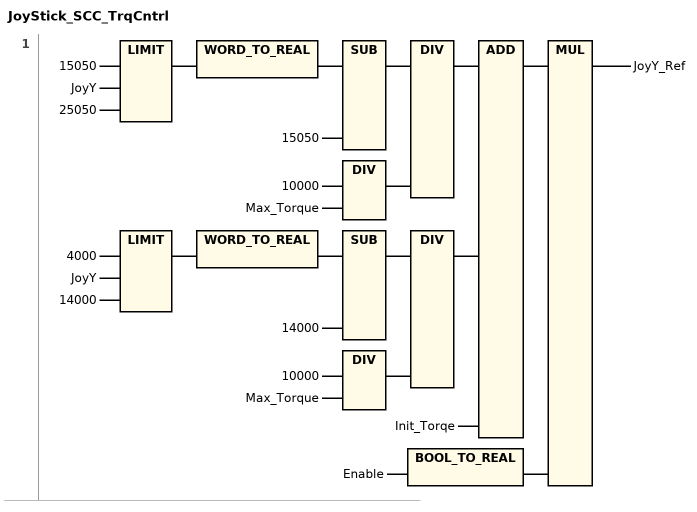
// NETWORK 1
JoyY_Ref := ((WORD_TO_REAL(LIMIT(15050, JoyY, 25050)) - 15050) / (10000 / Max_Torque) + (WORD_TO_REAL(LIMIT(4000, JoyY, 14000)) - 14000) / (10000 / Max_Torque) + Init_Torqe) * BOOL_TO_REAL(Enable);

END_FUNCTION_BLOCK

// IndraMotionMlc1/Application/VCC
PROGRAM VCC
VAR
	Enable_Motion_VCC_0: Enable_Motion_VCC;
	uValve: REAL := 6.0;
	JoyOut: REAL;
	ValveActive: BOOL;
	uValveMin: REAL := 3.0;
	uValveMax: REAL := 9.0;
	ActualValveOpening: REAL;
	uActualValveOpening: REAL;
	CylinderVelocity: REAL;
	
Ref: LREAL;
	InPosTime: LREAL;
	JerkRef: LREAL;
	Vel_Ref: LREAL := 0.0;
	Pos_Ref: LREAL := 0.0;
	uSignal: REAL := 6.0;
	ErrorSignal: LREAL;
	ManualMode: BOOL;
	uCtrl: REAL := 6.0;
	Reset: LREAL := 0.0;
	JoyOutDown: REAL;
	kFF: REAL;
	kFFdown: REAL;
	kFFup: REAL := 0.00275;
	Dist: LREAL := 450;
	VelSpV: LREAL := 50;
	

Sp: LREAL := 50;
	kCylRatio: REAL := 1.9;
	kP: LREAL := 0.0075;
	kI: LREAL := 0.001;
	MaxError: REAL := 1.0;
	MinError: REAL := -1.0;
	ZeroSignal: REAL := 6.0;
	Power_On: BOOL;
	JoyStick_VCC_0: JoyStick_VCC;
	ActValveOpening: REAL;
	VCC_PI_Controller_0: VCC_PI_Controller;
    uTest: REAL;
	uController: REAL;
	uManual: REAL;
END_VAR
VAR // added by the converter: edge detectors and wires of the graphical bodies
    _w1, _w2 : INT;
END_VAR

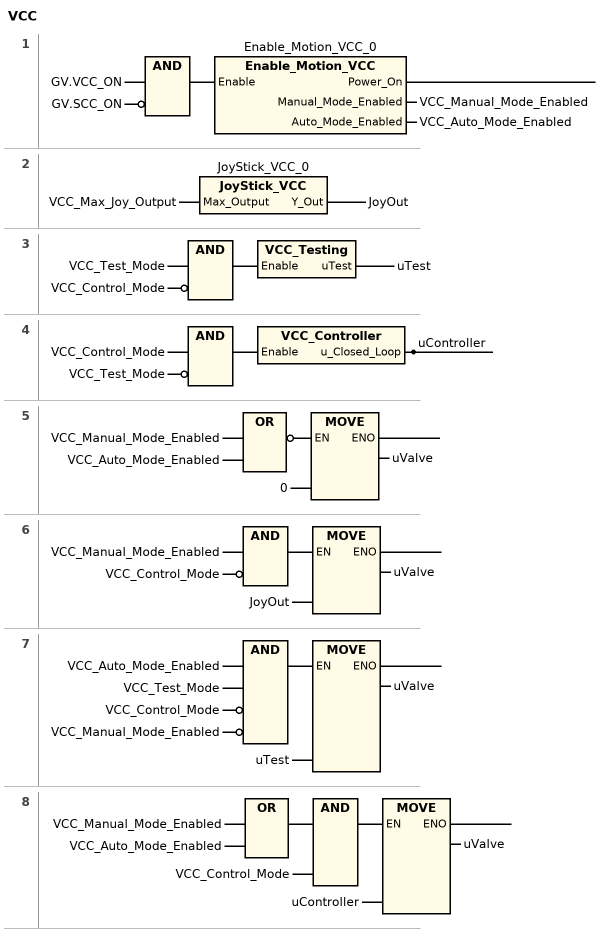
// NETWORK 1
Enable_Motion_VCC_0(
    Enable := GV.VCC_ON AND NOT GV.SCC_ON,
    Manual_Mode_Enabled => VCC_Manual_Mode_Enabled,
    Auto_Mode_Enabled => VCC_Auto_Mode_Enabled); // Enable_Motion_VCC

// NETWORK 2
JoyStick_VCC_0(Max_Output := VCC_Max_Joy_Output); // JoyStick_VCC
JoyOut := JoyStick_VCC_0.Y_Out;

// NETWORK 3
VCC_Testing(Enable := VCC_Test_Mode AND NOT VCC_Control_Mode);
uTest := VCC_Testing.uTest;

// NETWORK 4
VCC_Controller(Enable := VCC_Control_Mode AND NOT VCC_Test_Mode, u_Closed_Loop => uController);

// NETWORK 5
IF NOT (VCC_Manual_Mode_Enabled OR VCC_Auto_Mode_Enabled) THEN uValve := 0; END_IF

// NETWORK 6
IF VCC_Manual_Mode_Enabled AND NOT VCC_Control_Mode THEN uValve := JoyOut; END_IF

// NETWORK 7
IF VCC_Auto_Mode_Enabled AND VCC_Test_Mode AND NOT VCC_Control_Mode AND NOT VCC_Manual_Mode_Enabled THEN
    uValve := uTest;
END_IF

// NETWORK 8
IF (VCC_Manual_Mode_Enabled OR VCC_Auto_Mode_Enabled) AND VCC_Control_Mode THEN uValve := uController; END_IF

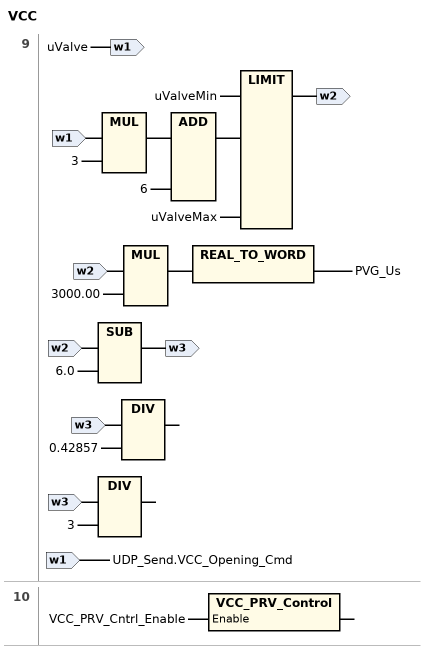
// NETWORK 9
_w1 := LIMIT(uValveMin, uValve * 3 + 6, uValveMax);
PVG_Us := REAL_TO_WORD(_w1 * 3000.00);
_w2 := _w1 - 6.0;
(* _w2 / 0.42857; result not used *)
(* _w2 / 3; result not used *)
UDP_Send.VCC_Opening_Cmd := uValve;

// NETWORK 10
VCC_PRV_Control(Enable := VCC_PRV_Cntrl_Enable);

END_PROGRAM

// IndraMotionMlc1/Application/Enable_Motion_VCC
FUNCTION_BLOCK Enable_Motion_VCC
VAR_INPUT
	Enable: BOOL;
END_VAR
VAR_OUTPUT
	 Power_On: BOOL;
	 Manual_Mode_Enabled: BOOL;
	 Auto_Mode_Enabled: BOOL;
END_VAR
VAR
	GreenLight: SR;
END_VAR
VAR // added by the converter: edge detectors and wires of the graphical bodies
    _w1 : BOOL;
END_VAR

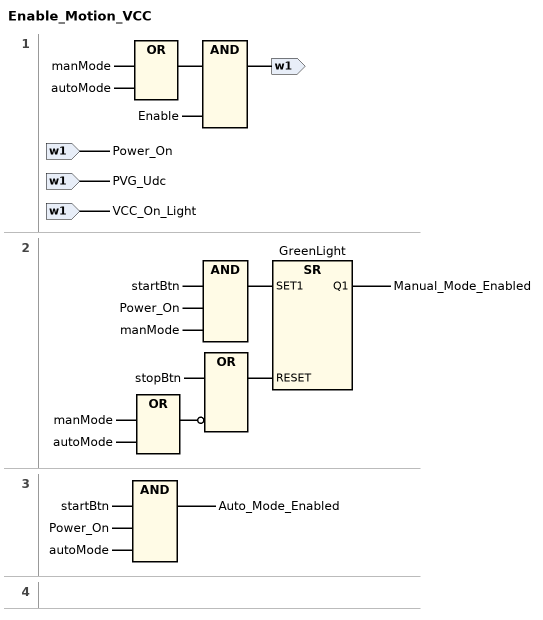
// NETWORK 1
_w1 := (manMode OR autoMode) AND Enable;
Power_On := _w1;
PVG_Udc := _w1;
VCC_On_Light := _w1;

// NETWORK 2
GreenLight(SET1 := startBtn AND Power_On AND manMode, RESET := stopBtn OR NOT (manMode OR autoMode)); // SR
Manual_Mode_Enabled := GreenLight.Q1;

// NETWORK 3
Auto_Mode_Enabled := startBtn AND Power_On AND autoMode;

// NETWORK 4

END_FUNCTION_BLOCK

// IndraMotionMlc1/Application/JoyStick_VCC
FUNCTION_BLOCK JoyStick_VCC
VAR_INPUT
	Max_Output: REAL := 100.0;
END_VAR
VAR_OUTPUT
	Y_Out: REAL;
END_VAR

VAR

END_VAR

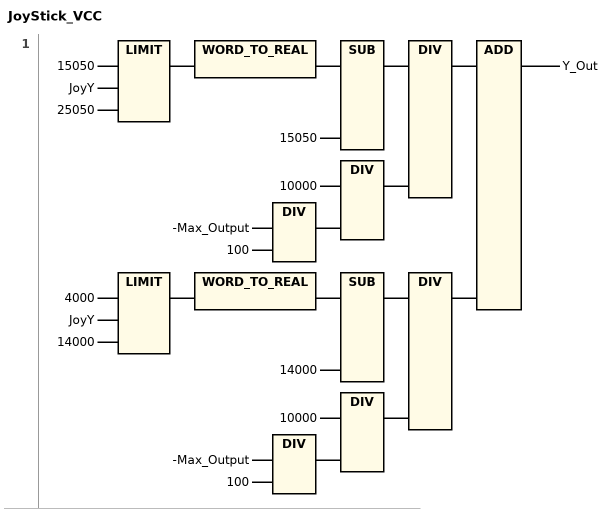
// NETWORK 1
Y_Out := (WORD_TO_REAL(LIMIT(15050, JoyY, 25050)) - 15050) / (10000 / ((-Max_Output) / 100)) + (WORD_TO_REAL(LIMIT(4000, JoyY, 14000)) - 14000) / (10000 / ((-Max_Output) / 100));

END_FUNCTION_BLOCK

// IndraMotionMlc1/Application/VCC_Testing
PROGRAM VCC_Testing
VAR_INPUT
	Enable: BOOL;
END_VAR


VAR
	VCC_StepFunction_Test_0: VCC_StepFunction_Test;	
	SinuousCurve_Test_0: SinuousCurve_Test;
	Ramp_Test_0: Ramp_Test;
	uStep: REAL;
	t0_Step: LREAL; 
	t1_Step: LREAL;
	t2_Step: LREAL;
	t3_Step: LREAL;

	uSin: REAL;
	t0_Sin: LREAL;
	T_test_Sin: LREAL := 10;
	f_Sin: LREAL := 0.1;
	uRamp: REAL;
	tHold_Up_Up_Up_ramp: LREAL := 1;
	tWait_ramp: LREAL := 4;
	uExt: LREAL;
	uRetr: LREAL;
	VCC_Anti_Dead_Band_v2_0: VCC_Anti_Dead_Band_v2;
	Ramp_Test_1: Ramp_Test;
	VCC_StepFunction_0: VCC_StepFunction;
	up_down: LREAL;
	VCC_Step_Function_Validation_0: VCC_Step_Function_Validation;
	uSP: LREAL;
	DB: LREAL;
	uPF: LREAL;
	PF2_0: PF2;
	VCC_Anti_Dead_Band_v2_1: VCC_Anti_Dead_Band_v2;
	JoyStick_VCC_0: JoyStick_VCC;
	uPF_Test: REAL;
	PF1_0: PF1;
	uPF1: LREAL;
	uPF2: LREAL;
	uPF11: LREAL;
	uPF_Test_DB: REAL;
	uPF_Joy: REAL;
	uJoy: REAL;
	uLPPF: LREAL;
	uStep_ref: LREAL;
	HPPF_pB_0: HPPF_pB;
	uPF_pB: LREAL;
	HPPF2_pB_0: HPPF2_pB;
	uPF_pB_vInfOFF: LREAL;
	uPF_pB_vInfOn: LREAL;
	uPF_pL: LREAL;
	HPPF_pA_0: HPPF_pA;
	uPF_pA: LREAL;
	HPPF2_pA_0: HPPF2_pA;
	uPF_pA_vInfOn: LREAL;
	uPF_pA_vInfOff: LREAL;
END_VAR

VAR_OUTPUT
	uTest: REAL;	
END_VAR
VAR // added by the converter: edge detectors and wires of the graphical bodies
    _w1, _w2, _w3, _w4, _w5, _w6, _w7 : BOOL;
END_VAR

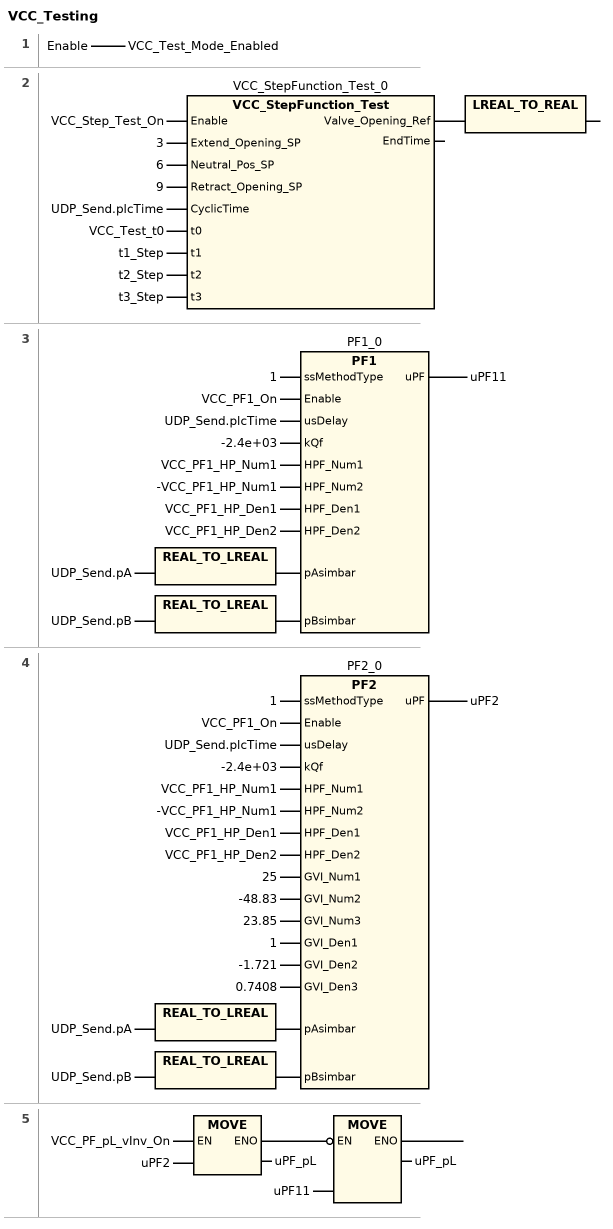
// NETWORK 1
VCC_Test_Mode_Enabled := Enable;

// NETWORK 2
VCC_StepFunction_Test_0(
    Enable := VCC_Step_Test_On,
    Extend_Opening_SP := 3,
    Neutral_Pos_SP := 6,
    Retract_Opening_SP := 9,
    CyclicTime := UDP_Send.plcTime,
    t0 := VCC_Test_t0,
    t1 := t1_Step,
    t2 := t2_Step,
    t3 := t3_Step); // VCC_StepFunction_Test
LREAL_TO_REAL(VCC_StepFunction_Test_0.Valve_Opening_Ref);

// NETWORK 3
PF1_0(
    ssMethodType := 1,
    Enable := VCC_PF1_On,
    usDelay := UDP_Send.plcTime,
    kQf := -2.4e+03,
    HPF_Num1 := VCC_PF1_HP_Num1,
    HPF_Num2 := -VCC_PF1_HP_Num1,
    HPF_Den1 := VCC_PF1_HP_Den1,
    HPF_Den2 := VCC_PF1_HP_Den2,
    pAsimbar := REAL_TO_LREAL(UDP_Send.pA),
    pBsimbar := REAL_TO_LREAL(UDP_Send.pB)); // PF1
uPF11 := PF1_0.uPF;

// NETWORK 4
PF2_0(
    ssMethodType := 1,
    Enable := VCC_PF1_On,
    usDelay := UDP_Send.plcTime,
    kQf := -2.4e+03,
    HPF_Num1 := VCC_PF1_HP_Num1,
    HPF_Num2 := -VCC_PF1_HP_Num1,
    HPF_Den1 := VCC_PF1_HP_Den1,
    HPF_Den2 := VCC_PF1_HP_Den2,
    GVI_Num1 := 25,
    GVI_Num2 := -48.83,
    GVI_Num3 := 23.85,
    GVI_Den1 := 1,
    GVI_Den2 := -1.721,
    GVI_Den3 := 0.7408,
    pAsimbar := REAL_TO_LREAL(UDP_Send.pA),
    pBsimbar := REAL_TO_LREAL(UDP_Send.pB)); // PF2
uPF2 := PF2_0.uPF;

// NETWORK 5
_w1 := VCC_PF_pL_vInv_On;
IF _w1 THEN uPF_pL := uPF2; END_IF
IF NOT _w1 THEN uPF_pL := uPF11; END_IF

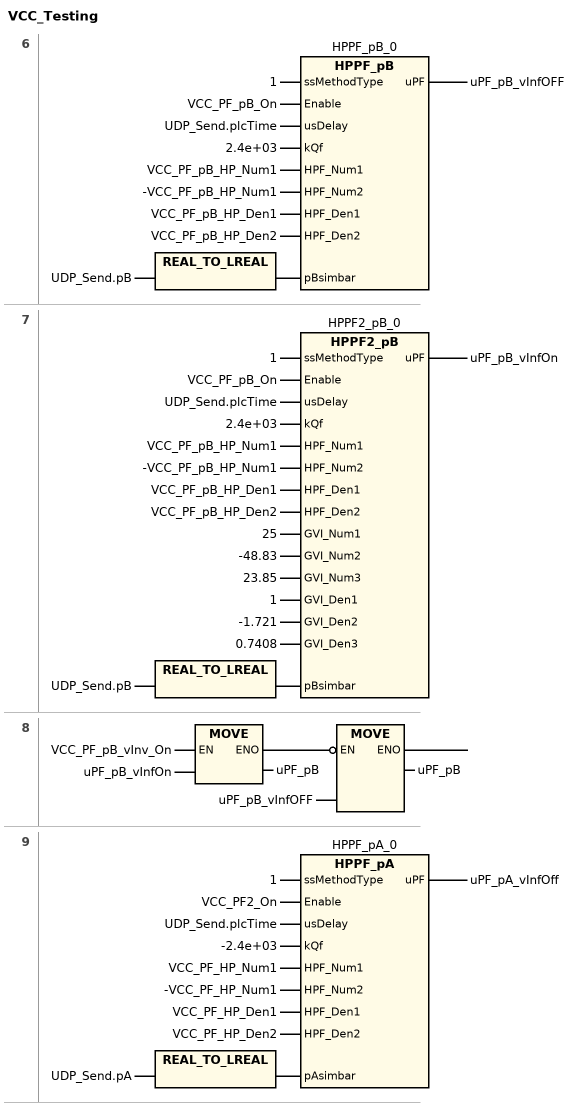
// NETWORK 6
HPPF_pB_0(
    ssMethodType := 1,
    Enable := VCC_PF_pB_On,
    usDelay := UDP_Send.plcTime,
    kQf := 2.4e+03,
    HPF_Num1 := VCC_PF_pB_HP_Num1,
    HPF_Num2 := -VCC_PF_pB_HP_Num1,
    HPF_Den1 := VCC_PF_pB_HP_Den1,
    HPF_Den2 := VCC_PF_pB_HP_Den2,
    pBsimbar := REAL_TO_LREAL(UDP_Send.pB)); // HPPF_pB
uPF_pB_vInfOFF := HPPF_pB_0.uPF;

// NETWORK 7
HPPF2_pB_0(
    ssMethodType := 1,
    Enable := VCC_PF_pB_On,
    usDelay := UDP_Send.plcTime,
    kQf := 2.4e+03,
    HPF_Num1 := VCC_PF_pB_HP_Num1,
    HPF_Num2 := -VCC_PF_pB_HP_Num1,
    HPF_Den1 := VCC_PF_pB_HP_Den1,
    HPF_Den2 := VCC_PF_pB_HP_Den2,
    GVI_Num1 := 25,
    GVI_Num2 := -48.83,
    GVI_Num3 := 23.85,
    GVI_Den1 := 1,
    GVI_Den2 := -1.721,
    GVI_Den3 := 0.7408,
    pBsimbar := REAL_TO_LREAL(UDP_Send.pB)); // HPPF2_pB
uPF_pB_vInfOn := HPPF2_pB_0.uPF;

// NETWORK 8
_w2 := VCC_PF_pB_vInv_On;
IF _w2 THEN uPF_pB := uPF_pB_vInfOn; END_IF
IF NOT _w2 THEN uPF_pB := uPF_pB_vInfOFF; END_IF

// NETWORK 9
HPPF_pA_0(
    ssMethodType := 1,
    Enable := VCC_PF2_On,
    usDelay := UDP_Send.plcTime,
    kQf := -2.4e+03,
    HPF_Num1 := VCC_PF_HP_Num1,
    HPF_Num2 := -VCC_PF_HP_Num1,
    HPF_Den1 := VCC_PF_HP_Den1,
    HPF_Den2 := VCC_PF_HP_Den2,
    pAsimbar := REAL_TO_LREAL(UDP_Send.pA)); // HPPF_pA
uPF_pA_vInfOff := HPPF_pA_0.uPF;

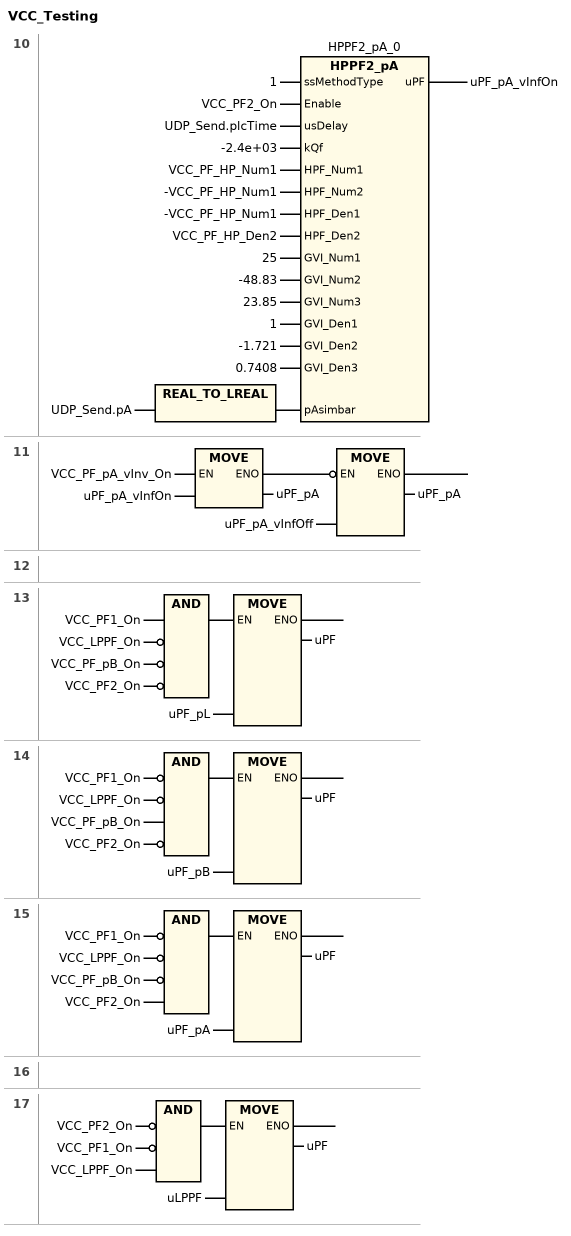
// NETWORK 10
HPPF2_pA_0(
    ssMethodType := 1,
    Enable := VCC_PF2_On,
    usDelay := UDP_Send.plcTime,
    kQf := -2.4e+03,
    HPF_Num1 := VCC_PF_HP_Num1,
    HPF_Num2 := -VCC_PF_HP_Num1,
    HPF_Den1 := -VCC_PF_HP_Num1,
    HPF_Den2 := VCC_PF_HP_Den2,
    GVI_Num1 := 25,
    GVI_Num2 := -48.83,
    GVI_Num3 := 23.85,
    GVI_Den1 := 1,
    GVI_Den2 := -1.721,
    GVI_Den3 := 0.7408,
    pAsimbar := REAL_TO_LREAL(UDP_Send.pA)); // HPPF2_pA
uPF_pA_vInfOn := HPPF2_pA_0.uPF;

// NETWORK 11
_w3 := VCC_PF_pA_vInv_On;
IF _w3 THEN uPF_pA := uPF_pA_vInfOn; END_IF
IF NOT _w3 THEN uPF_pA := uPF_pA_vInfOff; END_IF

// NETWORK 12

// NETWORK 13
IF VCC_PF1_On AND NOT VCC_LPPF_On AND NOT VCC_PF_pB_On AND NOT VCC_PF2_On THEN uPF := uPF_pL; END_IF

// NETWORK 14
IF NOT VCC_PF1_On AND NOT VCC_LPPF_On AND VCC_PF_pB_On AND NOT VCC_PF2_On THEN uPF := uPF_pB; END_IF

// NETWORK 15
IF NOT VCC_PF1_On AND NOT VCC_LPPF_On AND NOT VCC_PF_pB_On AND VCC_PF2_On THEN uPF := uPF_pA; END_IF

// NETWORK 16

// NETWORK 17
IF NOT VCC_PF2_On AND NOT VCC_PF1_On AND VCC_LPPF_On THEN uPF := uLPPF; END_IF

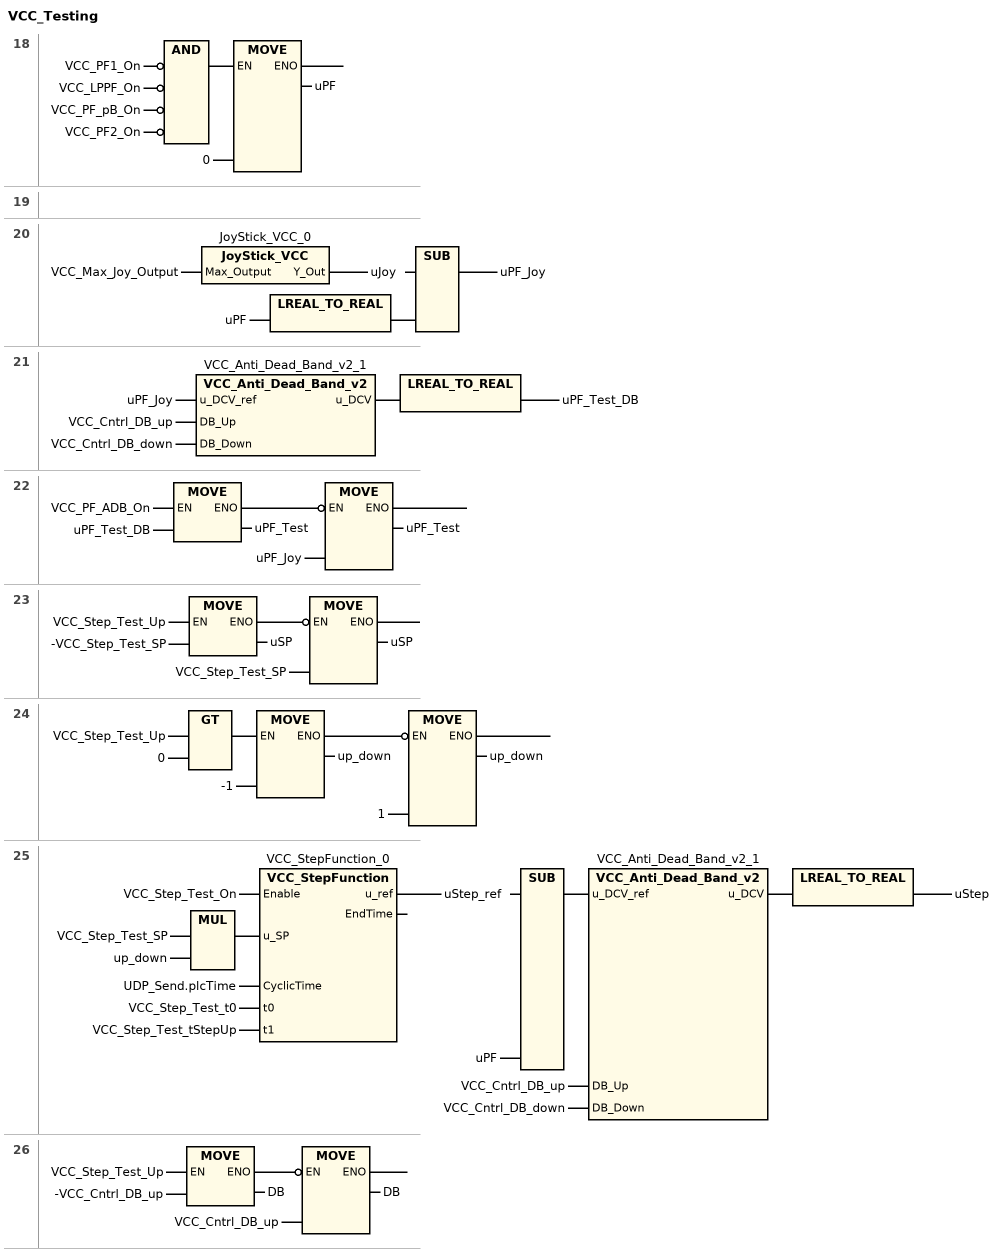
// NETWORK 18
IF NOT VCC_PF1_On AND NOT VCC_LPPF_On AND NOT VCC_PF_pB_On AND NOT VCC_PF2_On THEN uPF := 0; END_IF

// NETWORK 19

// NETWORK 20
JoyStick_VCC_0(Max_Output := VCC_Max_Joy_Output); // JoyStick_VCC
uJoy := JoyStick_VCC_0.Y_Out;
uPF_Joy := JoyStick_VCC_0.Y_Out - LREAL_TO_REAL(uPF);

// NETWORK 21
VCC_Anti_Dead_Band_v2_1(u_DCV_ref := uPF_Joy, DB_Up := VCC_Cntrl_DB_up, DB_Down := VCC_Cntrl_DB_down); // VCC_Anti_Dead_Band_v2
uPF_Test_DB := LREAL_TO_REAL(VCC_Anti_Dead_Band_v2_1.u_DCV);

// NETWORK 22
_w4 := VCC_PF_ADB_On;
IF _w4 THEN uPF_Test := uPF_Test_DB; END_IF
IF NOT _w4 THEN uPF_Test := uPF_Joy; END_IF

// NETWORK 23
_w5 := VCC_Step_Test_Up;
IF _w5 THEN uSP := -VCC_Step_Test_SP; END_IF
IF NOT _w5 THEN uSP := VCC_Step_Test_SP; END_IF

// NETWORK 24
_w6 := VCC_Step_Test_Up > 0;
IF _w6 THEN up_down := -1; END_IF
IF NOT _w6 THEN up_down := 1; END_IF

// NETWORK 25
VCC_StepFunction_0(
    Enable := VCC_Step_Test_On,
    u_SP := VCC_Step_Test_SP * up_down,
    CyclicTime := UDP_Send.plcTime,
    t0 := VCC_Step_Test_t0,
    t1 := VCC_Step_Test_tStepUp); // VCC_StepFunction
uStep_ref := VCC_StepFunction_0.u_ref;
VCC_Anti_Dead_Band_v2_1(
    u_DCV_ref := VCC_StepFunction_0.u_ref - uPF,
    DB_Up := VCC_Cntrl_DB_up,
    DB_Down := VCC_Cntrl_DB_down); // VCC_Anti_Dead_Band_v2
uStep := LREAL_TO_REAL(VCC_Anti_Dead_Band_v2_1.u_DCV);

// NETWORK 26
_w7 := VCC_Step_Test_Up;
IF _w7 THEN DB := -VCC_Cntrl_DB_up; END_IF
IF NOT _w7 THEN DB := VCC_Cntrl_DB_up; END_IF

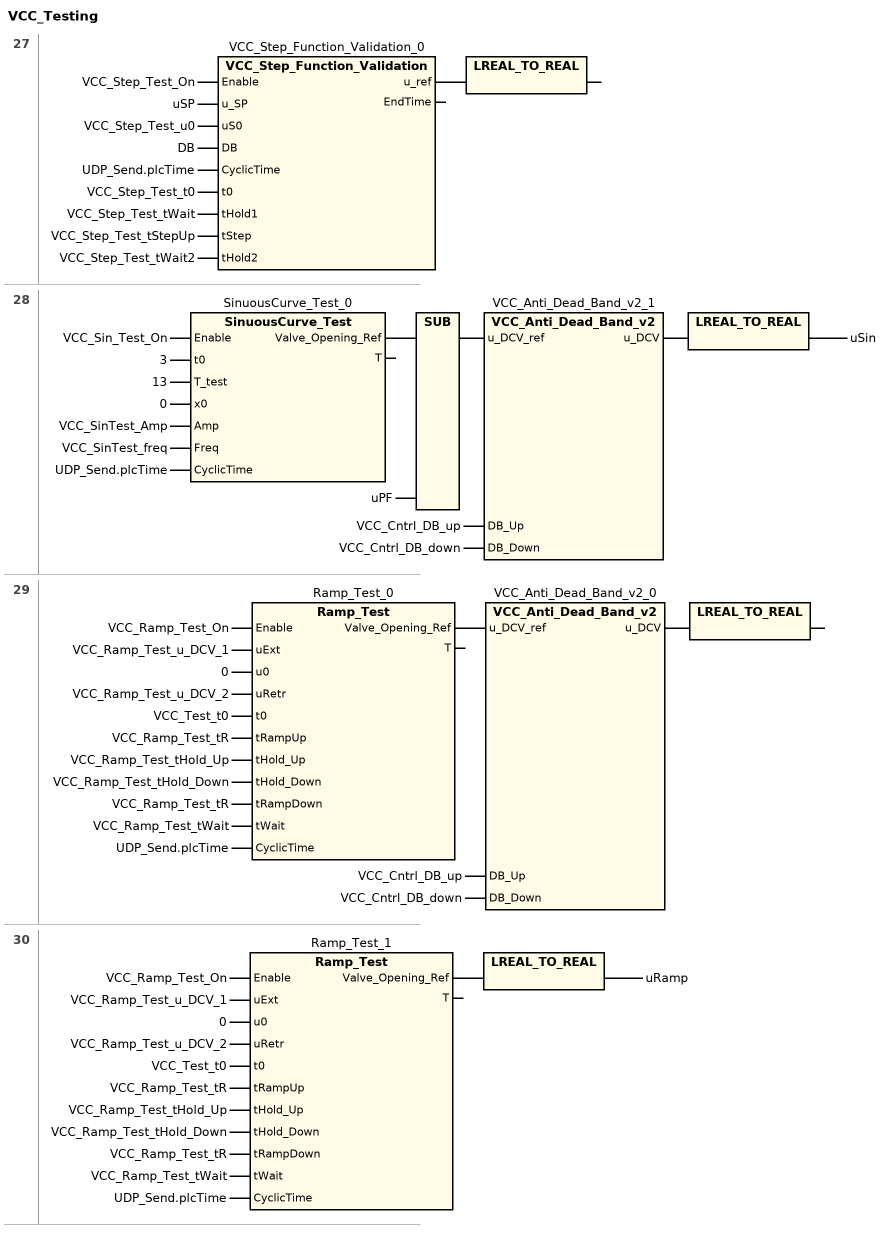
// NETWORK 27
VCC_Step_Function_Validation_0(
    Enable := VCC_Step_Test_On,
    u_SP := uSP,
    uS0 := VCC_Step_Test_u0,
    DB := DB,
    CyclicTime := UDP_Send.plcTime,
    t0 := VCC_Step_Test_t0,
    tHold1 := VCC_Step_Test_tWait,
    tStep := VCC_Step_Test_tStepUp,
    tHold2 := VCC_Step_Test_tWait2); // VCC_Step_Function_Validation
LREAL_TO_REAL(VCC_Step_Function_Validation_0.u_ref);

// NETWORK 28
SinuousCurve_Test_0(
    Enable := VCC_Sin_Test_On,
    t0 := 3,
    T_test := 13,
    x0 := 0,
    Amp := VCC_SinTest_Amp,
    Freq := VCC_SinTest_freq,
    CyclicTime := UDP_Send.plcTime); // SinuousCurve_Test
VCC_Anti_Dead_Band_v2_1(
    u_DCV_ref := SinuousCurve_Test_0.Valve_Opening_Ref - uPF,
    DB_Up := VCC_Cntrl_DB_up,
    DB_Down := VCC_Cntrl_DB_down); // VCC_Anti_Dead_Band_v2
uSin := LREAL_TO_REAL(VCC_Anti_Dead_Band_v2_1.u_DCV);

